ABB RAPID module: 000EB206

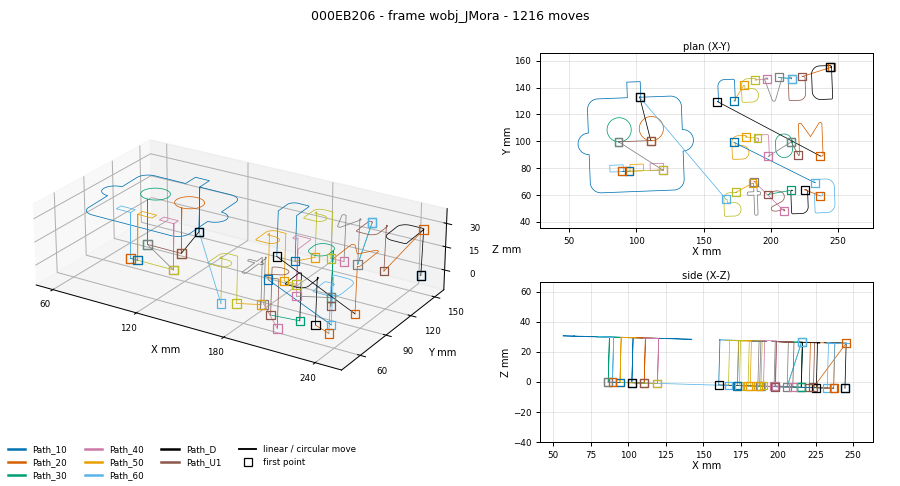
[picture p0: tool path of 000EB206 in frame wobj_JMora, 1216 of 1225 moves have a stored position in this frame; points joined in program order, loops and branches not executed]
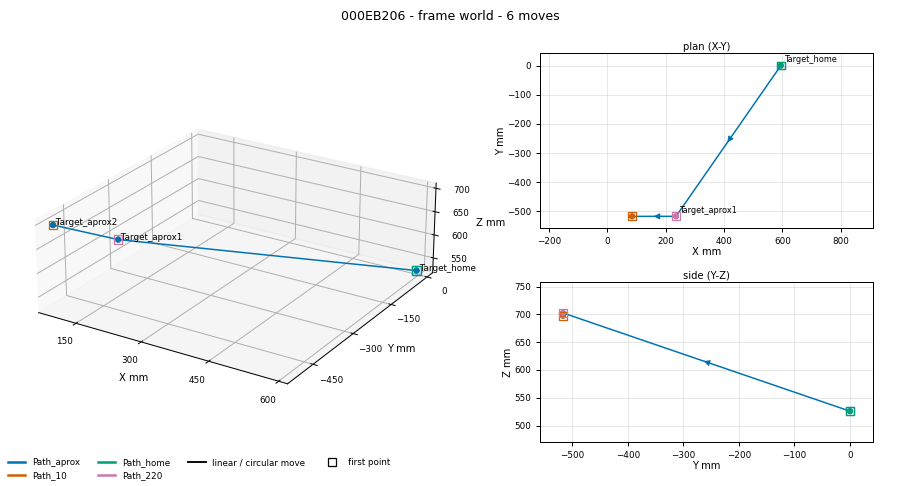
[picture p1: tool path of 000EB206 in frame world, 6 of 1225 moves have a stored position in this frame; points joined in program order, loops and branches not executed]
MODULE Module1
	PERS tooldata toolreal_fin:=[TRUE,[[75.2786,-1.94785,145.188],[1,0,0,0]],[1,[0,0,0],[1,0,0,0],0,0,0]];
    TASK PERS tooldata toolreal:=[TRUE,[[0,0,0],[1,0,0,0]],[-1,[0,0,0],[1,0,0,0],0,0,0]];

    CONST robtarget Target_home:=[[594.991189092,-0.007598177,525.862524879],[0.258822484,0.000002114,0.965924905,-0.000003007],[0,0,0,0],[9E+09,9E+09,9E+09,9E+09,9E+09,9E+09]];
    CONST robtarget Target_aprox1:=[[235.86399401,-516.605376424,702.653598227],[0,0.707106781,0.707106781,0],[0,0,0,0],[9E+09,9E+09,9E+09,9E+09,9E+09,9E+09]];
    CONST robtarget Target_aprox2:=[[85.598000009,-516.640000054,697.650000033],[0,0.707106781,0.707106781,0],[0,0,0,0],[9E+09,9E+09,9E+09,9E+09,9E+09,9E+09]];
    CONST robtarget Target_10:=[[244.458254265,155.289204222,-4.164726397],[0.692516726,0.060687774,-0.040025667,0.717729422],[-2,0,-1,0],[9E+09,9E+09,9E+09,9E+09,9E+09,9E+09]];
    CONST robtarget Target_20:=[[245.259577842,155.215414434,25.824478921],[0.692516726,0.060687774,-0.040025667,0.717729422],[-2,0,-1,0],[9E+09,9E+09,9E+09,9E+09,9E+09,9E+09]];
    CONST robtarget Target_30:=[[245.229089406,155.507196472,25.826011527],[0.692516726,0.060687774,-0.040025667,0.717729422],[-2,0,-1,0],[9E+09,9E+09,9E+09,9E+09,9E+09,9E+09]];
    CONST robtarget Target_40:=[[245.16107836,155.758507333,25.82844716],[0.692516726,0.060687774,-0.040025666,0.717729422],[-2,0,-1,0],[9E+09,9E+09,9E+09,9E+09,9E+09,9E+09]];
    CONST robtarget Target_50:=[[245.055544704,155.969347015,25.831785853],[0.692516726,0.060687774,-0.040025667,0.717729422],[-2,0,-1,0],[9E+09,9E+09,9E+09,9E+09,9E+09,9E+09]];
    CONST robtarget Target_60:=[[244.912488436,156.139715523,25.836027573],[0.692516726,0.060687774,-0.040025667,0.717729422],[-2,0,-1,0],[9E+09,9E+09,9E+09,9E+09,9E+09,9E+09]];
    CONST robtarget Target_70:=[[244.73190956,156.269612854,25.841172332],[0.692516726,0.060687774,-0.040025667,0.717729422],[-2,0,-1,0],[9E+09,9E+09,9E+09,9E+09,9E+09,9E+09]];
    CONST robtarget Target_80:=[[244.513808072,156.359039007,25.847220128],[0.692516726,0.060687774,-0.040025667,0.717729422],[-2,0,-1,0],[9E+09,9E+09,9E+09,9E+09,9E+09,9E+09]];
    CONST robtarget Target_90:=[[244.258183973,156.407993984,25.854170962],[0.692516726,0.060687774,-0.040025667,0.717729422],[-2,0,-1,0],[9E+09,9E+09,9E+09,9E+09,9E+09,9E+09]];
    CONST robtarget Target_100:=[[243.965037266,156.416477784,25.862024834],[0.692516726,0.060687774,-0.040025667,0.717729422],[-2,0,-1,0],[9E+09,9E+09,9E+09,9E+09,9E+09,9E+09]];
    CONST robtarget Target_110:=[[236.458451079,156.133651424,26.061907917],[0.692516726,0.060687774,-0.040025667,0.717729422],[-1,-1,0,0],[9E+09,9E+09,9E+09,9E+09,9E+09,9E+09]];
    CONST robtarget Target_120:=[[235.817178284,156.081173489,26.078913847],[0.692516726,0.060687774,-0.040025666,0.717729422],[-1,-1,0,0],[9E+09,9E+09,9E+09,9E+09,9E+09,9E+09]];
    CONST robtarget Target_130:=[[235.20337356,155.973097192,26.09504904],[0.692516726,0.060687774,-0.040025667,0.717729422],[-1,-1,0,0],[9E+09,9E+09,9E+09,9E+09,9E+09,9E+09]];
    CONST robtarget Target_140:=[[234.617036903,155.809422533,26.11031345],[0.692516726,0.060687774,-0.040025666,0.717729422],[-1,-1,0,0],[9E+09,9E+09,9E+09,9E+09,9E+09,9E+09]];
    CONST robtarget Target_150:=[[234.058168316,155.590149513,26.124707111],[0.692516726,0.060687774,-0.040025666,0.717729422],[-1,-1,0,0],[9E+09,9E+09,9E+09,9E+09,9E+09,9E+09]];
    CONST robtarget Target_160:=[[233.526767795,155.315278129,26.138230024],[0.692516726,0.060687774,-0.040025667,0.717729422],[-1,-1,0,0],[9E+09,9E+09,9E+09,9E+09,9E+09,9E+09]];
    CONST robtarget Target_170:=[[233.022835345,154.984808384,26.150882165],[0.692516726,0.060687774,-0.040025667,0.717729422],[-1,-1,0,0],[9E+09,9E+09,9E+09,9E+09,9E+09,9E+09]];
    CONST robtarget Target_180:=[[232.546370963,154.598740279,26.162663546],[0.692516726,0.060687774,-0.040025667,0.717729422],[-1,-1,0,0],[9E+09,9E+09,9E+09,9E+09,9E+09,9E+09]];
    CONST robtarget Target_190:=[[232.097374649,154.157073811,26.173574156],[0.692516726,0.060687774,-0.040025666,0.717729422],[-1,-1,0,0],[9E+09,9E+09,9E+09,9E+09,9E+09,9E+09]];
    CONST robtarget Target_200:=[[231.690855447,153.675997451,26.183252813],[0.692516726,0.060687774,-0.040025667,0.717729422],[-1,-1,0,0],[9E+09,9E+09,9E+09,9E+09,9E+09,9E+09]];
    CONST robtarget Target_210:=[[231.341822403,153.171699671,26.191338269],[0.692516726,0.060687774,-0.040025667,0.717729422],[-1,-1,0,0],[9E+09,9E+09,9E+09,9E+09,9E+09,9E+09]];
    CONST robtarget Target_220:=[[231.050275515,152.644180472,26.197830522],[0.692516726,0.060687774,-0.040025666,0.717729422],[-1,-1,0,0],[9E+09,9E+09,9E+09,9E+09,9E+09,9E+09]];
    CONST robtarget Target_230:=[[230.816214785,152.093439851,26.202729597],[0.692516726,0.060687774,-0.040025666,0.717729422],[-1,-1,0,0],[9E+09,9E+09,9E+09,9E+09,9E+09,9E+09]];
    CONST robtarget Target_240:=[[230.639640211,151.519477809,26.206035481],[0.692516726,0.060687774,-0.040025666,0.717729422],[-1,-1,0,0],[9E+09,9E+09,9E+09,9E+09,9E+09,9E+09]];
    CONST robtarget Target_250:=[[230.520551793,150.922294347,26.207748185],[0.692516726,0.060687774,-0.040025667,0.717729422],[-1,-1,0,0],[9E+09,9E+09,9E+09,9E+09,9E+09,9E+09]];
    CONST robtarget Target_260:=[[230.458949533,150.301889466,26.207867677],[0.692516726,0.060687774,-0.040025666,0.717729422],[-1,-1,0,0],[9E+09,9E+09,9E+09,9E+09,9E+09,9E+09]];
    CONST robtarget Target_270:=[[230.45483343,149.658263163,26.206394001],[0.692516726,0.060687774,-0.040025667,0.717729422],[-1,-1,0,0],[9E+09,9E+09,9E+09,9E+09,9E+09,9E+09]];
    CONST robtarget Target_280:=[[230.924700472,137.156756977,26.163078447],[0.692516726,0.060687774,-0.040025667,0.717729422],[-1,-1,0,0],[9E+09,9E+09,9E+09,9E+09,9E+09,9E+09]];
    CONST robtarget Target_290:=[[230.977088342,136.52469846,26.160123414],[0.692516726,0.060687774,-0.040025667,0.717729422],[-1,-1,0,0],[9E+09,9E+09,9E+09,9E+09,9E+09,9E+09]];
    CONST robtarget Target_300:=[[231.085779815,135.918195759,26.155726818],[0.692516726,0.060687774,-0.040025666,0.717729422],[-1,-1,0,0],[9E+09,9E+09,9E+09,9E+09,9E+09,9E+09]];
    CONST robtarget Target_310:=[[231.250774887,135.337248876,26.149888616],[0.692516726,0.060687774,-0.040025666,0.717729422],[-1,-1,0,0],[9E+09,9E+09,9E+09,9E+09,9E+09,9E+09]];
    CONST robtarget Target_320:=[[231.472073561,134.781857808,26.142608862],[0.692516726,0.060687774,-0.040025666,0.717729422],[-1,-1,0,0],[9E+09,9E+09,9E+09,9E+09,9E+09,9E+09]];
    CONST robtarget Target_330:=[[231.749675836,134.252022554,26.133887545],[0.692516726,0.060687774,-0.040025667,0.717729422],[-1,-1,0,0],[9E+09,9E+09,9E+09,9E+09,9E+09,9E+09]];
    CONST robtarget Target_340:=[[232.083581711,133.747743119,26.123724645],[0.692516726,0.060687774,-0.040025667,0.717729422],[-1,-1,0,0],[9E+09,9E+09,9E+09,9E+09,9E+09,9E+09]];
    CONST robtarget Target_350:=[[232.473791188,133.2690195,26.112120159],[0.692516726,0.060687774,-0.040025666,0.717729422],[-1,-1,0,0],[9E+09,9E+09,9E+09,9E+09,9E+09,9E+09]];
    CONST robtarget Target_360:=[[232.920304265,132.815851696,26.099074122],[0.692516726,0.060687774,-0.040025667,0.717729422],[-1,-1,0,0],[9E+09,9E+09,9E+09,9E+09,9E+09,9E+09]];
    CONST robtarget Target_370:=[[233.405590707,132.40450411,26.085094935],[0.692516726,0.060687774,-0.040025667,0.717729422],[-1,-1,0,0],[9E+09,9E+09,9E+09,9E+09,9E+09,9E+09]];
    CONST robtarget Target_380:=[[233.912120276,132.051241138,26.070691042],[0.692516726,0.060687774,-0.040025667,0.717729422],[-1,-1,0,0],[9E+09,9E+09,9E+09,9E+09,9E+09,9E+09]];
    CONST robtarget Target_390:=[[234.439892972,131.756062782,26.055862424],[0.692516726,0.060687774,-0.040025667,0.717729422],[-1,-1,0,0],[9E+09,9E+09,9E+09,9E+09,9E+09,9E+09]];
    CONST robtarget Target_400:=[[234.988908794,131.518969041,26.040609121],[0.692516726,0.060687774,-0.040025667,0.717729422],[-1,-1,0,0],[9E+09,9E+09,9E+09,9E+09,9E+09,9E+09]];
    CONST robtarget Target_410:=[[235.559167743,131.339959914,26.024931135],[0.692516726,0.060687774,-0.040025667,0.717729422],[-1,-1,0,0],[9E+09,9E+09,9E+09,9E+09,9E+09,9E+09]];
    CONST robtarget Target_420:=[[236.15066982,131.219035404,26.008828422],[0.692516726,0.060687774,-0.040025667,0.717729422],[-1,-1,0,0],[9E+09,9E+09,9E+09,9E+09,9E+09,9E+09]];
    CONST robtarget Target_430:=[[236.763415023,131.156195509,25.992301005],[0.692516726,0.060687774,-0.040025667,0.717729422],[-1,-1,0,0],[9E+09,9E+09,9E+09,9E+09,9E+09,9E+09]];
    CONST robtarget Target_440:=[[237.397403355,131.151440229,25.975348882],[0.692516726,0.060687774,-0.040025667,0.717729422],[-1,-1,0,0],[9E+09,9E+09,9E+09,9E+09,9E+09,9E+09]];
    CONST robtarget Target_530:=[[246.104713071,132.729344243,25.746568583],[0.692516726,0.060687774,-0.040025667,0.717729422],[-2,0,-1,0],[9E+09,9E+09,9E+09,9E+09,9E+09,9E+09]];
    CONST robtarget Target_510:=[[246.047258547,132.180375453,25.746753017],[0.692516726,0.060687774,-0.040025666,0.717729422],[-2,0,-1,0],[9E+09,9E+09,9E+09,9E+09,9E+09,9E+09]];
    CONST robtarget Target_520:=[[246.096213006,132.436093232,25.746074151],[0.692516726,0.060687774,-0.040025667,0.717729422],[-2,0,-1,0],[9E+09,9E+09,9E+09,9E+09,9E+09,9E+09]];
    CONST robtarget Target_540:=[[245.259577842,155.215414434,25.824478921],[0.692516726,0.060687774,-0.040025667,0.717729422],[-2,0,-1,0],[9E+09,9E+09,9E+09,9E+09,9E+09,9E+09]];
    CONST robtarget Target_500:=[[245.957849696,131.9621909,25.748605216],[0.692516726,0.060687774,-0.040025667,0.717729422],[-2,0,-1,0],[9E+09,9E+09,9E+09,9E+09,9E+09,9E+09]];
    CONST robtarget Target_450:=[[244.903989542,131.43426659,25.7754658],[0.692516726,0.060687774,-0.040025667,0.717729422],[-2,0,-1,0],[9E+09,9E+09,9E+09,9E+09,9E+09,9E+09]];
    CONST robtarget Target_460:=[[245.195670358,131.464784994,25.767747052],[0.692516726,0.060687774,-0.040025666,0.717729422],[-2,0,-1,0],[9E+09,9E+09,9E+09,9E+09,9E+09,9E+09]];
    CONST robtarget Target_480:=[[245.657668813,131.638421488,25.75582952],[0.692516726,0.060687774,-0.040025667,0.717729422],[-2,0,-1,0],[9E+09,9E+09,9E+09,9E+09,9E+09,9E+09]];
    CONST robtarget Target_490:=[[245.827986451,131.78153958,25.751630702],[0.692516726,0.060687774,-0.040025666,0.717729422],[-2,0,-1,0],[9E+09,9E+09,9E+09,9E+09,9E+09,9E+09]];
    CONST robtarget Target_470:=[[245.446896782,131.532836625,25.761201637],[0.692516726,0.060687774,-0.040025667,0.717729422],[-2,0,-1,0],[9E+09,9E+09,9E+09,9E+09,9E+09,9E+09]];
    CONST robtarget Target_550:=[[223.462258109,148.248946692,-3.621027841],[0.692516726,0.060687774,-0.040025667,0.717729422],[0,0,0,0],[9E+09,9E+09,9E+09,9E+09,9E+09,9E+09]];
    CONST robtarget Target_560:=[[224.263581686,148.175156905,26.368177477],[0.692516726,0.060687774,-0.040025667,0.717729422],[0,0,0,0],[9E+09,9E+09,9E+09,9E+09,9E+09,9E+09]];
    CONST robtarget Target_570:=[[224.556728395,148.166673106,26.360323594],[0.692516726,0.060687774,-0.040025666,0.717729422],[0,0,0,0],[9E+09,9E+09,9E+09,9E+09,9E+09,9E+09]];
    CONST robtarget Target_580:=[[224.812352494,148.117718127,26.353372782],[0.692516726,0.060687774,-0.040025666,0.717729422],[0,0,0,0],[9E+09,9E+09,9E+09,9E+09,9E+09,9E+09]];
    CONST robtarget Target_590:=[[225.03045398,148.028291975,26.347324964],[0.692516726,0.060687774,-0.040025666,0.717729422],[0,0,0,0],[9E+09,9E+09,9E+09,9E+09,9E+09,9E+09]];
    CONST robtarget Target_600:=[[225.211032857,147.898394643,26.342180217],[0.692516726,0.060687774,-0.040025667,0.717729422],[0,0,0,0],[9E+09,9E+09,9E+09,9E+09,9E+09,9E+09]];
    CONST robtarget Target_610:=[[225.354089124,147.728026137,26.337938485],[0.692516726,0.060687774,-0.040025666,0.717729422],[0,0,0,0],[9E+09,9E+09,9E+09,9E+09,9E+09,9E+09]];
    CONST robtarget Target_620:=[[225.459622781,147.517186454,26.334599803],[0.692516726,0.060687774,-0.040025666,0.717729422],[0,0,0,0],[9E+09,9E+09,9E+09,9E+09,9E+09,9E+09]];
    CONST robtarget Target_630:=[[225.527633827,147.265875592,26.33216417],[0.692516726,0.060687774,-0.040025667,0.717729422],[0,0,0,0],[9E+09,9E+09,9E+09,9E+09,9E+09,9E+09]];
    CONST robtarget Target_640:=[[225.558122263,146.974093555,26.330631564],[0.692516726,0.060687774,-0.040025667,0.717729422],[0,0,0,0],[9E+09,9E+09,9E+09,9E+09,9E+09,9E+09]];
    CONST robtarget Target_650:=[[225.981080782,135.720657872,26.291640359],[0.692516726,0.060687774,-0.040025667,0.717729422],[0,0,0,0],[9E+09,9E+09,9E+09,9E+09,9E+09,9E+09]];
    CONST robtarget Target_660:=[[225.977855815,135.204815501,26.290457267],[0.692516726,0.060687774,-0.040025666,0.717729422],[0,0,0,0],[9E+09,9E+09,9E+09,9E+09,9E+09,9E+09]];
    CONST robtarget Target_670:=[[225.928699575,134.707747724,26.290547695],[0.692516726,0.060687774,-0.040025667,0.717729422],[0,0,0,0],[9E+09,9E+09,9E+09,9E+09,9E+09,9E+09]];
    CONST robtarget Target_680:=[[225.833612059,134.229454546,26.291911598],[0.692516726,0.060687774,-0.040025666,0.717729422],[0,0,0,0],[9E+09,9E+09,9E+09,9E+09,9E+09,9E+09]];
    CONST robtarget Target_690:=[[225.69259327,133.769935961,26.294549011],[0.692516726,0.060687774,-0.040025666,0.717729422],[0,0,0,0],[9E+09,9E+09,9E+09,9E+09,9E+09,9E+09]];
    CONST robtarget Target_700:=[[225.505643208,133.329191973,26.298459921],[0.692516726,0.060687774,-0.040025666,0.717729422],[0,0,0,0],[9E+09,9E+09,9E+09,9E+09,9E+09,9E+09]];
    CONST robtarget Target_710:=[[225.272761871,132.907222579,26.30364434],[0.692516726,0.060687774,-0.040025667,0.717729422],[0,0,0,0],[9E+09,9E+09,9E+09,9E+09,9E+09,9E+09]];
    CONST robtarget Target_720:=[[224.99394926,132.504027783,26.310102235],[0.692516726,0.060687774,-0.040025666,0.717729422],[0,0,0,0],[9E+09,9E+09,9E+09,9E+09,9E+09,9E+09]];
    CONST robtarget Target_730:=[[224.669205374,132.119607582,26.317833638],[0.692516726,0.060687774,-0.040025666,0.717729422],[0,0,0,0],[9E+09,9E+09,9E+09,9E+09,9E+09,9E+09]];
    CONST robtarget Target_740:=[[224.310412375,131.766777849,26.326552577],[0.692516726,0.060687774,-0.040025666,0.717729422],[0,0,0,0],[9E+09,9E+09,9E+09,9E+09,9E+09,9E+09]];
    CONST robtarget Target_750:=[[223.929452421,131.458354456,26.33597309],[0.692516726,0.060687774,-0.040025666,0.717729422],[0,0,0,0],[9E+09,9E+09,9E+09,9E+09,9E+09,9E+09]];
    CONST robtarget Target_760:=[[223.526325513,131.194337404,26.346095188],[0.692516726,0.060687774,-0.040025667,0.717729422],[0,0,0,0],[9E+09,9E+09,9E+09,9E+09,9E+09,9E+09]];
    CONST robtarget Target_770:=[[223.101031652,130.974726695,26.356918848],[0.692516726,0.060687774,-0.040025667,0.717729422],[0,0,0,0],[9E+09,9E+09,9E+09,9E+09,9E+09,9E+09]];
    CONST robtarget Target_780:=[[222.653570836,130.799522325,26.368444082],[0.692516726,0.060687774,-0.040025667,0.717729422],[0,0,0,0],[9E+09,9E+09,9E+09,9E+09,9E+09,9E+09]];
    CONST robtarget Target_790:=[[222.183943066,130.668724296,26.38067089],[0.692516726,0.060687774,-0.040025667,0.717729422],[0,0,0,0],[9E+09,9E+09,9E+09,9E+09,9E+09,9E+09]];
    CONST robtarget Target_800:=[[221.692148341,130.582332609,26.393599271],[0.692516726,0.060687774,-0.040025667,0.717729422],[0,0,0,0],[9E+09,9E+09,9E+09,9E+09,9E+09,9E+09]];
    CONST robtarget Target_810:=[[221.178186662,130.540347262,26.407229226],[0.692516726,0.060687774,-0.040025667,0.717729422],[0,0,0,0],[9E+09,9E+09,9E+09,9E+09,9E+09,9E+09]];
    CONST robtarget Target_820:=[[214.919232528,130.304528053,26.573890744],[0.692516726,0.060687774,-0.040025667,0.717729422],[0,0,0,0],[9E+09,9E+09,9E+09,9E+09,9E+09,9E+09]];
    CONST robtarget Target_830:=[[214.626085821,130.313011855,26.581744605],[0.692516726,0.060687774,-0.040025666,0.717729422],[0,0,0,0],[9E+09,9E+09,9E+09,9E+09,9E+09,9E+09]];
    CONST robtarget Target_840:=[[214.370461724,130.36196683,26.588695461],[0.692516726,0.060687774,-0.040025666,0.717729422],[0,0,0,0],[9E+09,9E+09,9E+09,9E+09,9E+09,9E+09]];
    CONST robtarget Target_850:=[[214.152360235,130.451392985,26.594743235],[0.692516726,0.060687774,-0.040025666,0.717729422],[0,0,0,0],[9E+09,9E+09,9E+09,9E+09,9E+09,9E+09]];
    CONST robtarget Target_860:=[[213.971781358,130.581290314,26.599888004],[0.692516726,0.060687774,-0.040025667,0.717729422],[0,0,0,0],[9E+09,9E+09,9E+09,9E+09,9E+09,9E+09]];
    CONST robtarget Target_870:=[[213.828725091,130.751658823,26.604129713],[0.692516726,0.060687774,-0.040025666,0.717729422],[0,0,0,0],[9E+09,9E+09,9E+09,9E+09,9E+09,9E+09]];
    CONST robtarget Target_880:=[[213.723191435,130.962498507,26.607468396],[0.692516726,0.060687774,-0.040025666,0.717729422],[0,0,0,0],[9E+09,9E+09,9E+09,9E+09,9E+09,9E+09]];
    CONST robtarget Target_890:=[[213.655180388,131.213809365,26.609904051],[0.692516726,0.060687774,-0.040025667,0.717729422],[0,0,0,0],[9E+09,9E+09,9E+09,9E+09,9E+09,9E+09]];
    CONST robtarget Target_900:=[[213.624691952,131.505591403,26.611436657],[0.692516726,0.060687774,-0.040025667,0.717729422],[0,0,0,0],[9E+09,9E+09,9E+09,9E+09,9E+09,9E+09]];
    CONST robtarget Target_910:=[[213.061007863,146.503238589,26.663400906],[0.692516726,0.060687774,-0.040025667,0.717729422],[0,0,0,0],[9E+09,9E+09,9E+09,9E+09,9E+09,9E+09]];
    CONST robtarget Target_920:=[[213.069507929,146.796489599,26.663895338],[0.692516726,0.060687774,-0.040025667,0.717729422],[0,0,0,0],[9E+09,9E+09,9E+09,9E+09,9E+09,9E+09]];
    CONST robtarget Target_930:=[[213.118462388,147.052207381,26.66321645],[0.692516726,0.060687774,-0.040025666,0.717729422],[0,0,0,0],[9E+09,9E+09,9E+09,9E+09,9E+09,9E+09]];
    CONST robtarget Target_940:=[[213.207871239,147.270391931,26.661364273],[0.692516726,0.060687774,-0.040025667,0.717729422],[0,0,0,0],[9E+09,9E+09,9E+09,9E+09,9E+09,9E+09]];
    CONST robtarget Target_950:=[[213.337734484,147.451043254,26.658338765],[0.692516726,0.060687774,-0.040025666,0.717729422],[0,0,0,0],[9E+09,9E+09,9E+09,9E+09,9E+09,9E+09]];
    CONST robtarget Target_960:=[[213.508052121,147.594161345,26.654139969],[0.692516726,0.060687774,-0.040025667,0.717729422],[0,0,0,0],[9E+09,9E+09,9E+09,9E+09,9E+09,9E+09]];
    CONST robtarget Target_970:=[[213.718824152,147.699746206,26.648767852],[0.692516726,0.060687774,-0.040025667,0.717729422],[0,0,0,0],[9E+09,9E+09,9E+09,9E+09,9E+09,9E+09]];
    CONST robtarget Target_980:=[[213.970050576,147.76779784,26.642222415],[0.692516726,0.060687774,-0.040025666,0.717729422],[0,0,0,0],[9E+09,9E+09,9E+09,9E+09,9E+09,9E+09]];
    CONST robtarget Target_990:=[[214.261731393,147.798316241,26.634503689],[0.692516726,0.060687774,-0.040025667,0.717729422],[0,0,0,0],[9E+09,9E+09,9E+09,9E+09,9E+09,9E+09]];
    CONST robtarget Target_1000:=[[214.554878101,147.789832442,26.626649806],[0.692516726,0.060687774,-0.040025666,0.717729422],[0,0,0,0],[9E+09,9E+09,9E+09,9E+09,9E+09,9E+09]];
    CONST robtarget Target_1010:=[[214.8105022,147.740877464,26.619698994],[0.692516726,0.060687774,-0.040025666,0.717729422],[0,0,0,0],[9E+09,9E+09,9E+09,9E+09,9E+09,9E+09]];
    CONST robtarget Target_1020:=[[215.028603686,147.651451311,26.613651176],[0.692516726,0.060687774,-0.040025666,0.717729422],[0,0,0,0],[9E+09,9E+09,9E+09,9E+09,9E+09,9E+09]];
    CONST robtarget Target_1030:=[[215.209182564,147.52155398,26.608506429],[0.692516726,0.060687774,-0.040025667,0.717729422],[0,0,0,0],[9E+09,9E+09,9E+09,9E+09,9E+09,9E+09]];
    CONST robtarget Target_1040:=[[215.35223883,147.351185473,26.604264698],[0.692516726,0.060687774,-0.040025666,0.717729422],[0,0,0,0],[9E+09,9E+09,9E+09,9E+09,9E+09,9E+09]];
    CONST robtarget Target_1050:=[[215.457772487,147.14034579,26.600926016],[0.692516726,0.060687774,-0.040025666,0.717729422],[0,0,0,0],[9E+09,9E+09,9E+09,9E+09,9E+09,9E+09]];
    CONST robtarget Target_1060:=[[215.525783533,146.889034929,26.598490382],[0.692516726,0.060687774,-0.040025667,0.717729422],[0,0,0,0],[9E+09,9E+09,9E+09,9E+09,9E+09,9E+09]];
    CONST robtarget Target_1070:=[[215.55627197,146.597252891,26.596957776],[0.692516726,0.060687774,-0.040025667,0.717729422],[0,0,0,0],[9E+09,9E+09,9E+09,9E+09,9E+09,9E+09]];
    CONST robtarget Target_1080:=[[205.974615496,147.590063121,-3.155372239],[0.692516726,0.060687774,-0.040025667,0.717729422],[0,0,0,0],[9E+09,9E+09,9E+09,9E+09,9E+09,9E+09]];
    CONST robtarget Target_1090:=[[206.775939073,147.516273333,26.833833079],[0.692516726,0.060687774,-0.040025667,0.717729422],[0,0,0,0],[9E+09,9E+09,9E+09,9E+09,9E+09,9E+09]];
    CONST robtarget Target_1100:=[[207.018522887,147.502629685,26.827317561],[0.692516726,0.060687774,-0.040025666,0.717729422],[0,0,0,0],[9E+09,9E+09,9E+09,9E+09,9E+09,9E+09]];
    CONST robtarget Target_1110:=[[207.247221507,147.442895875,26.821059664],[0.692516726,0.060687774,-0.040025666,0.717729422],[0,0,0,0],[9E+09,9E+09,9E+09,9E+09,9E+09,9E+09]];
    CONST robtarget Target_1120:=[[207.462034933,147.337071905,26.815059401],[0.692516726,0.060687774,-0.040025666,0.717729422],[0,0,0,0],[9E+09,9E+09,9E+09,9E+09,9E+09,9E+09]];
    CONST robtarget Target_1130:=[[207.662963164,147.185157777,26.809316704],[0.692516726,0.060687774,-0.040025666,0.717729422],[0,0,0,0],[9E+09,9E+09,9E+09,9E+09,9E+09,9E+09]];
    CONST robtarget Target_1140:=[[207.833873307,147.000866706,26.804296471],[0.692516726,0.060687774,-0.040025667,0.717729422],[0,0,0,0],[9E+09,9E+09,9E+09,9E+09,9E+09,9E+09]];
    CONST robtarget Target_1150:=[[207.958632467,146.797911914,26.800463466],[0.692516726,0.060687774,-0.040025666,0.717729422],[0,0,0,0],[9E+09,9E+09,9E+09,9E+09,9E+09,9E+09]];
    CONST robtarget Target_1160:=[[208.037240646,146.576293398,26.797817744],[0.692516726,0.060687774,-0.040025666,0.717729422],[0,0,0,0],[9E+09,9E+09,9E+09,9E+09,9E+09,9E+09]];
    CONST robtarget Target_1170:=[[208.069697841,146.336011159,26.796359239],[0.692516726,0.060687774,-0.040025667,0.717729422],[0,0,0,0],[9E+09,9E+09,9E+09,9E+09,9E+09,9E+09]];
    CONST robtarget Target_1180:=[[208.056331156,146.137616545,26.796228232],[0.692516726,0.060687774,-0.040025666,0.717729422],[0,0,0,0],[9E+09,9E+09,9E+09,9E+09,9E+09,9E+09]];
    CONST robtarget Target_1190:=[[208.002158545,145.91685385,26.797132549],[0.692516726,0.060687774,-0.040025666,0.717729422],[0,0,0,0],[9E+09,9E+09,9E+09,9E+09,9E+09,9E+09]];
    CONST robtarget Target_1200:=[[203.652235422,130.900721267,26.876416368],[0.692516726,0.060687774,-0.040025666,0.717729422],[0,0,0,0],[9E+09,9E+09,9E+09,9E+09,9E+09,9E+09]];
    CONST robtarget Target_1210:=[[203.564392561,130.658184821,26.878166804],[0.692516726,0.060687774,-0.040025667,0.717729422],[0,0,0,0],[9E+09,9E+09,9E+09,9E+09,9E+09,9E+09]];
    CONST robtarget Target_1220:=[[203.458457537,130.44686362,26.880477464],[0.692516726,0.060687774,-0.040025667,0.717729422],[0,0,0,0],[9E+09,9E+09,9E+09,9E+09,9E+09,9E+09]];
    CONST robtarget Target_1230:=[[203.334430353,130.266757664,26.883348351],[0.692516726,0.060687774,-0.040025666,0.717729422],[0,0,0,0],[9E+09,9E+09,9E+09,9E+09,9E+09,9E+09]];
    CONST robtarget Target_1240:=[[203.192311005,130.11786695,26.886779495],[0.692516726,0.060687774,-0.040025667,0.717729422],[0,0,0,0],[9E+09,9E+09,9E+09,9E+09,9E+09,9E+09]];
    CONST robtarget Target_1250:=[[203.032099496,130.000191481,26.890770865],[0.692516726,0.060687774,-0.040025667,0.717729422],[0,0,0,0],[9E+09,9E+09,9E+09,9E+09,9E+09,9E+09]];
    CONST robtarget Target_1260:=[[202.853795825,129.913731256,26.895322471],[0.692516726,0.060687774,-0.040025667,0.717729422],[0,0,0,0],[9E+09,9E+09,9E+09,9E+09,9E+09,9E+09]];
    CONST robtarget Target_1270:=[[202.657399992,129.858486276,26.900434314],[0.692516726,0.060687774,-0.040025667,0.717729422],[0,0,0,0],[9E+09,9E+09,9E+09,9E+09,9E+09,9E+09]];
    CONST robtarget Target_1280:=[[202.442911997,129.834456539,26.906106393],[0.692516726,0.060687774,-0.040025667,0.717729422],[0,0,0,0],[9E+09,9E+09,9E+09,9E+09,9E+09,9E+09]];
    CONST robtarget Target_1290:=[[202.222341078,129.84242,26.91201972],[0.692516726,0.060687774,-0.040025666,0.717729422],[0,0,0,0],[9E+09,9E+09,9E+09,9E+09,9E+09,9E+09]];
    CONST robtarget Target_1300:=[[202.018093409,129.883546331,26.917578503],[0.692516726,0.060687774,-0.040025667,0.717729422],[0,0,0,0],[9E+09,9E+09,9E+09,9E+09,9E+09,9E+09]];
    CONST robtarget Target_1310:=[[201.830168991,129.95783554,26.9227827],[0.692516726,0.060687774,-0.040025666,0.717729422],[0,0,0,0],[9E+09,9E+09,9E+09,9E+09,9E+09,9E+09]];
    CONST robtarget Target_1320:=[[201.658567821,130.065287622,26.927632343],[0.692516726,0.060687774,-0.040025666,0.717729422],[0,0,0,0],[9E+09,9E+09,9E+09,9E+09,9E+09,9E+09]];
    CONST robtarget Target_1330:=[[201.503289901,130.205902577,26.93212742],[0.692516726,0.060687774,-0.040025666,0.717729422],[0,0,0,0],[9E+09,9E+09,9E+09,9E+09,9E+09,9E+09]];
    CONST robtarget Target_1340:=[[201.364335231,130.379680405,26.936267944],[0.692516726,0.060687774,-0.040025667,0.717729422],[0,0,0,0],[9E+09,9E+09,9E+09,9E+09,9E+09,9E+09]];
    CONST robtarget Target_1350:=[[201.24170381,130.586621109,26.940053891],[0.692516726,0.060687774,-0.040025667,0.717729422],[0,0,0,0],[9E+09,9E+09,9E+09,9E+09,9E+09,9E+09]];
    CONST robtarget Target_1360:=[[201.135395639,130.826724686,26.943485274],[0.692516726,0.060687774,-0.040025667,0.717729422],[0,0,0,0],[9E+09,9E+09,9E+09,9E+09,9E+09,9E+09]];
    CONST robtarget Target_1370:=[[195.671395086,145.452266503,27.12547236],[0.692516726,0.060687774,-0.040025667,0.717729422],[0,0,0,0],[9E+09,9E+09,9E+09,9E+09,9E+09,9E+09]];
    CONST robtarget Target_1380:=[[195.600804491,145.668328483,27.127890199],[0.692516726,0.060687774,-0.040025667,0.717729422],[0,0,0,0],[9E+09,9E+09,9E+09,9E+09,9E+09,9E+09]];
    CONST robtarget Target_1390:=[[195.572583442,145.865156193,27.129128581],[0.692516726,0.060687774,-0.040025667,0.717729422],[0,0,0,0],[9E+09,9E+09,9E+09,9E+09,9E+09,9E+09]];
    CONST robtarget Target_1400:=[[195.581591648,146.153544169,27.129597469],[0.692516726,0.060687774,-0.040025667,0.717729422],[0,0,0,0],[9E+09,9E+09,9E+09,9E+09,9E+09,9E+09]];
    CONST robtarget Target_1410:=[[195.631679624,146.405073435,27.128877998],[0.692516726,0.060687774,-0.040025667,0.717729422],[0,0,0,0],[9E+09,9E+09,9E+09,9E+09,9E+09,9E+09]];
    CONST robtarget Target_1420:=[[195.722847369,146.619743992,27.126970165],[0.692516726,0.060687774,-0.040025667,0.717729422],[0,0,0,0],[9E+09,9E+09,9E+09,9E+09,9E+09,9E+09]];
    CONST robtarget Target_1430:=[[195.855094885,146.79755584,27.123873962],[0.692516726,0.060687774,-0.040025666,0.717729422],[0,0,0,0],[9E+09,9E+09,9E+09,9E+09,9E+09,9E+09]];
    CONST robtarget Target_1440:=[[196.028422171,146.938508975,27.11958942],[0.692516726,0.060687774,-0.040025667,0.717729422],[0,0,0,0],[9E+09,9E+09,9E+09,9E+09,9E+09,9E+09]];
    CONST robtarget Target_1450:=[[196.242829227,147.0426034,27.114116507],[0.692516726,0.060687774,-0.040025667,0.717729422],[0,0,0,0],[9E+09,9E+09,9E+09,9E+09,9E+09,9E+09]];
    CONST robtarget Target_1460:=[[196.498316052,147.109839116,27.107455233],[0.692516726,0.060687774,-0.040025667,0.717729422],[0,0,0,0],[9E+09,9E+09,9E+09,9E+09,9E+09,9E+09]];
    CONST robtarget Target_1470:=[[196.794882648,147.140216122,27.099605599],[0.692516726,0.060687774,-0.040025667,0.717729422],[0,0,0,0],[9E+09,9E+09,9E+09,9E+09,9E+09,9E+09]];
    CONST robtarget Target_1480:=[[197.014368912,147.135141106,27.093728339],[0.692516726,0.060687774,-0.040025666,0.717729422],[0,0,0,0],[9E+09,9E+09,9E+09,9E+09,9E+09,9E+09]];
    CONST robtarget Target_1490:=[[197.215362618,147.102680093,27.088277857],[0.692516726,0.060687774,-0.040025666,0.717729422],[0,0,0,0],[9E+09,9E+09,9E+09,9E+09,9E+09,9E+09]];
    CONST robtarget Target_1500:=[[197.397863764,147.042833091,27.083254086],[0.692516726,0.060687774,-0.040025667,0.717729422],[0,0,0,0],[9E+09,9E+09,9E+09,9E+09,9E+09,9E+09]];
    CONST robtarget Target_1510:=[[197.561872353,146.955600097,27.078657059],[0.692516726,0.060687774,-0.040025666,0.717729422],[0,0,0,0],[9E+09,9E+09,9E+09,9E+09,9E+09,9E+09]];
    CONST robtarget Target_1520:=[[197.707388383,146.840981108,27.074486799],[0.692516726,0.060687774,-0.040025667,0.717729422],[0,0,0,0],[9E+09,9E+09,9E+09,9E+09,9E+09,9E+09]];
    CONST robtarget Target_1530:=[[197.834411855,146.69897613,27.07074326],[0.692516726,0.060687774,-0.040025666,0.717729422],[0,0,0,0],[9E+09,9E+09,9E+09,9E+09,9E+09,9E+09]];
    CONST robtarget Target_1540:=[[197.942942768,146.529585157,27.067426487],[0.692516726,0.060687774,-0.040025667,0.717729422],[0,0,0,0],[9E+09,9E+09,9E+09,9E+09,9E+09,9E+09]];
    CONST robtarget Target_1550:=[[198.032981123,146.332808193,27.064536448],[0.692516726,0.060687774,-0.040025667,0.717729422],[0,0,0,0],[9E+09,9E+09,9E+09,9E+09,9E+09,9E+09]];
    CONST robtarget Target_1560:=[[197.231657546,146.406597981,-2.92466887],[0.692516726,0.060687774,-0.040025667,0.717729422],[0,0,0,0],[9E+09,9E+09,9E+09,9E+09,9E+09,9E+09]];
    CONST robtarget Target_1570:=[[188.51308754,145.682325596,-2.693487292],[0.692516726,0.060687774,-0.040025667,0.717729422],[0,0,0,0],[9E+09,9E+09,9E+09,9E+09,9E+09,9E+09]];
    CONST robtarget Target_1580:=[[189.314411117,145.608535808,27.295718026],[0.692516726,0.060687774,-0.040025667,0.717729422],[0,0,0,0],[9E+09,9E+09,9E+09,9E+09,9E+09,9E+09]];
    CONST robtarget Target_1590:=[[189.28392268,145.900317845,27.297250632],[0.692516726,0.060687774,-0.040025667,0.717729422],[0,0,0,0],[9E+09,9E+09,9E+09,9E+09,9E+09,9E+09]];
    CONST robtarget Target_1600:=[[189.215911634,146.151628707,27.299686265],[0.692516726,0.060687774,-0.040025666,0.717729422],[0,0,0,0],[9E+09,9E+09,9E+09,9E+09,9E+09,9E+09]];
    CONST robtarget Target_1610:=[[189.110377977,146.36246839,27.303024947],[0.692516726,0.060687774,-0.040025666,0.717729422],[0,0,0,0],[9E+09,9E+09,9E+09,9E+09,9E+09,9E+09]];
    CONST robtarget Target_1620:=[[188.96732171,146.532836896,27.307266678],[0.692516726,0.060687774,-0.040025667,0.717729422],[0,0,0,0],[9E+09,9E+09,9E+09,9E+09,9E+09,9E+09]];
    CONST robtarget Target_1630:=[[188.786742833,146.662734228,27.312411425],[0.692516726,0.060687774,-0.040025666,0.717729422],[0,0,0,0],[9E+09,9E+09,9E+09,9E+09,9E+09,9E+09]];
    CONST robtarget Target_1640:=[[188.568641346,146.75216038,27.318459243],[0.692516726,0.060687774,-0.040025666,0.717729422],[0,0,0,0],[9E+09,9E+09,9E+09,9E+09,9E+09,9E+09]];
    CONST robtarget Target_1650:=[[188.313017248,146.801115359,27.325410055],[0.692516726,0.060687774,-0.040025666,0.717729422],[0,0,0,0],[9E+09,9E+09,9E+09,9E+09,9E+09,9E+09]];
    CONST robtarget Target_1660:=[[188.01987054,146.809599158,27.333263939],[0.692516726,0.060687774,-0.040025667,0.717729422],[0,0,0,0],[9E+09,9E+09,9E+09,9E+09,9E+09,9E+09]];
    CONST robtarget Target_1670:=[[183.029342326,146.621570553,27.466150198],[0.692516726,0.060687774,-0.040025667,0.717729422],[0,0,0,0],[9E+09,9E+09,9E+09,9E+09,9E+09,9E+09]];
    CONST robtarget Target_1680:=[[182.515380648,146.579585206,27.479780153],[0.692516726,0.060687774,-0.040025667,0.717729422],[0,0,0,0],[9E+09,9E+09,9E+09,9E+09,9E+09,9E+09]];
    CONST robtarget Target_1690:=[[182.023585924,146.493193519,27.492708535],[0.692516726,0.060687774,-0.040025667,0.717729422],[0,0,0,0],[9E+09,9E+09,9E+09,9E+09,9E+09,9E+09]];
    CONST robtarget Target_1700:=[[181.553958153,146.36239549,27.504935342],[0.692516726,0.060687774,-0.040025667,0.717729422],[0,0,0,0],[9E+09,9E+09,9E+09,9E+09,9E+09,9E+09]];
    CONST robtarget Target_1710:=[[181.106497337,146.187191121,27.516460576],[0.692516726,0.060687774,-0.040025667,0.717729422],[0,0,0,0],[9E+09,9E+09,9E+09,9E+09,9E+09,9E+09]];
    CONST robtarget Target_1720:=[[180.681203475,145.967580411,27.527284237],[0.692516726,0.060687774,-0.040025667,0.717729422],[0,0,0,0],[9E+09,9E+09,9E+09,9E+09,9E+09,9E+09]];
    CONST robtarget Target_1730:=[[180.278076568,145.70356336,27.537406312],[0.692516726,0.060687774,-0.040025666,0.717729422],[0,0,0,0],[9E+09,9E+09,9E+09,9E+09,9E+09,9E+09]];
    CONST robtarget Target_1740:=[[179.897116615,145.395139968,27.546826825],[0.692516726,0.060687774,-0.040025666,0.717729422],[0,0,0,0],[9E+09,9E+09,9E+09,9E+09,9E+09,9E+09]];
    CONST robtarget Target_1750:=[[179.538323615,145.042310235,27.555545764],[0.692516726,0.060687774,-0.040025666,0.717729422],[0,0,0,0],[9E+09,9E+09,9E+09,9E+09,9E+09,9E+09]];
    CONST robtarget Target_1760:=[[179.21357973,144.657890034,27.563277168],[0.692516726,0.060687774,-0.040025666,0.717729422],[0,0,0,0],[9E+09,9E+09,9E+09,9E+09,9E+09,9E+09]];
    CONST robtarget Target_1770:=[[178.934767119,144.254695235,27.569735085],[0.692516726,0.060687774,-0.040025667,0.717729422],[0,0,0,0],[9E+09,9E+09,9E+09,9E+09,9E+09,9E+09]];
    CONST robtarget Target_1780:=[[178.701885782,143.832725843,27.574919482],[0.692516726,0.060687774,-0.040025666,0.717729422],[0,0,0,0],[9E+09,9E+09,9E+09,9E+09,9E+09,9E+09]];
    CONST robtarget Target_1790:=[[178.514935719,143.391981856,27.578830392],[0.692516726,0.060687774,-0.040025666,0.717729422],[0,0,0,0],[9E+09,9E+09,9E+09,9E+09,9E+09,9E+09]];
    CONST robtarget Target_1800:=[[178.373916929,142.932463271,27.581467804],[0.692516726,0.060687774,-0.040025666,0.717729422],[0,0,0,0],[9E+09,9E+09,9E+09,9E+09,9E+09,9E+09]];
    CONST robtarget Target_1810:=[[178.278829415,142.45417009,27.58283173],[0.692516726,0.060687774,-0.040025667,0.717729422],[0,0,0,0],[9E+09,9E+09,9E+09,9E+09,9E+09,9E+09]];
    CONST robtarget Target_1820:=[[178.229673174,141.957102316,27.582922136],[0.692516726,0.060687774,-0.040025666,0.717729422],[0,0,0,0],[9E+09,9E+09,9E+09,9E+09,9E+09,9E+09]];
    CONST robtarget Target_1830:=[[178.226448208,141.441259943,27.581739066],[0.692516726,0.060687774,-0.040025667,0.717729422],[0,0,0,0],[9E+09,9E+09,9E+09,9E+09,9E+09,9E+09]];
    CONST robtarget Target_1840:=[[178.649406727,130.18782426,27.54274786],[0.692516726,0.060687774,-0.040025667,0.717729422],[0,0,0,0],[9E+09,9E+09,9E+09,9E+09,9E+09,9E+09]];
    CONST robtarget Target_1850:=[[178.679895162,129.896042223,27.541215254],[0.692516726,0.060687774,-0.040025667,0.717729422],[0,0,0,0],[9E+09,9E+09,9E+09,9E+09,9E+09,9E+09]];
    CONST robtarget Target_1860:=[[178.747906209,129.644731364,27.538779599],[0.692516726,0.060687774,-0.040025666,0.717729422],[0,0,0,0],[9E+09,9E+09,9E+09,9E+09,9E+09,9E+09]];
    CONST robtarget Target_1870:=[[178.853439865,129.43389168,27.535440917],[0.692516726,0.060687774,-0.040025666,0.717729422],[0,0,0,0],[9E+09,9E+09,9E+09,9E+09,9E+09,9E+09]];
    CONST robtarget Target_1880:=[[178.996496132,129.263523172,27.531199208],[0.692516726,0.060687774,-0.040025667,0.717729422],[0,0,0,0],[9E+09,9E+09,9E+09,9E+09,9E+09,9E+09]];
    CONST robtarget Target_1890:=[[179.177075009,129.133625843,27.526054439],[0.692516726,0.060687774,-0.040025666,0.717729422],[0,0,0,0],[9E+09,9E+09,9E+09,9E+09,9E+09,9E+09]];
    CONST robtarget Target_1900:=[[179.395176498,129.044199688,27.520006665],[0.692516726,0.060687774,-0.040025666,0.717729422],[0,0,0,0],[9E+09,9E+09,9E+09,9E+09,9E+09,9E+09]];
    CONST robtarget Target_1910:=[[179.650800595,128.995244712,27.513055808],[0.692516726,0.060687774,-0.040025666,0.717729422],[0,0,0,0],[9E+09,9E+09,9E+09,9E+09,9E+09,9E+09]];
    CONST robtarget Target_1920:=[[179.943947303,128.98676091,27.505201947],[0.692516726,0.060687774,-0.040025667,0.717729422],[0,0,0,0],[9E+09,9E+09,9E+09,9E+09,9E+09,9E+09]];
    CONST robtarget Target_1930:=[[186.182107569,129.221796667,27.339094123],[0.692516726,0.060687774,-0.040025667,0.717729422],[0,0,0,0],[9E+09,9E+09,9E+09,9E+09,9E+09,9E+09]];
    CONST robtarget Target_1940:=[[186.696069248,129.263782014,27.325464167],[0.692516726,0.060687774,-0.040025667,0.717729422],[0,0,0,0],[9E+09,9E+09,9E+09,9E+09,9E+09,9E+09]];
    CONST robtarget Target_1950:=[[187.187863972,129.350173701,27.312535786],[0.692516726,0.060687774,-0.040025667,0.717729422],[0,0,0,0],[9E+09,9E+09,9E+09,9E+09,9E+09,9E+09]];
    CONST robtarget Target_1960:=[[187.657491742,129.48097173,27.300308978],[0.692516726,0.060687774,-0.040025667,0.717729422],[0,0,0,0],[9E+09,9E+09,9E+09,9E+09,9E+09,9E+09]];
    CONST robtarget Target_1970:=[[188.104952558,129.656176099,27.288783744],[0.692516726,0.060687774,-0.040025667,0.717729422],[0,0,0,0],[9E+09,9E+09,9E+09,9E+09,9E+09,9E+09]];
    CONST robtarget Target_1980:=[[188.530246421,129.875786809,27.277960084],[0.692516726,0.060687774,-0.040025667,0.717729422],[0,0,0,0],[9E+09,9E+09,9E+09,9E+09,9E+09,9E+09]];
    CONST robtarget Target_1990:=[[188.933373328,130.139803861,27.267837987],[0.692516726,0.060687774,-0.040025666,0.717729422],[0,0,0,0],[9E+09,9E+09,9E+09,9E+09,9E+09,9E+09]];
    CONST robtarget Target_2000:=[[189.314333281,130.448227253,27.258417474],[0.692516726,0.060687774,-0.040025666,0.717729422],[0,0,0,0],[9E+09,9E+09,9E+09,9E+09,9E+09,9E+09]];
    CONST robtarget Target_2010:=[[189.673126281,130.801056986,27.249698534],[0.692516726,0.060687774,-0.040025666,0.717729422],[0,0,0,0],[9E+09,9E+09,9E+09,9E+09,9E+09,9E+09]];
    CONST robtarget Target_2020:=[[189.997870166,131.185477188,27.241967131],[0.692516726,0.060687774,-0.040025666,0.717729422],[0,0,0,0],[9E+09,9E+09,9E+09,9E+09,9E+09,9E+09]];
    CONST robtarget Target_2030:=[[190.276682777,131.588671984,27.235509236],[0.692516726,0.060687774,-0.040025667,0.717729422],[0,0,0,0],[9E+09,9E+09,9E+09,9E+09,9E+09,9E+09]];
    CONST robtarget Target_2040:=[[190.509564114,132.010641378,27.230324817],[0.692516726,0.060687774,-0.040025666,0.717729422],[0,0,0,0],[9E+09,9E+09,9E+09,9E+09,9E+09,9E+09]];
    CONST robtarget Target_2050:=[[190.696514177,132.451385366,27.226413907],[0.692516726,0.060687774,-0.040025666,0.717729422],[0,0,0,0],[9E+09,9E+09,9E+09,9E+09,9E+09,9E+09]];
    CONST robtarget Target_2060:=[[190.837532966,132.91090395,27.223776495],[0.692516726,0.060687774,-0.040025666,0.717729422],[0,0,0,0],[9E+09,9E+09,9E+09,9E+09,9E+09,9E+09]];
    CONST robtarget Target_2070:=[[190.932620481,133.389197129,27.222412591],[0.692516726,0.060687774,-0.040025667,0.717729422],[0,0,0,0],[9E+09,9E+09,9E+09,9E+09,9E+09,9E+09]];
    CONST robtarget Target_2080:=[[190.981776722,133.886264906,27.222322163],[0.692516726,0.060687774,-0.040025666,0.717729422],[0,0,0,0],[9E+09,9E+09,9E+09,9E+09,9E+09,9E+09]];
    CONST robtarget Target_2090:=[[190.985001688,134.402107276,27.223505255],[0.692516726,0.060687774,-0.040025667,0.717729422],[0,0,0,0],[9E+09,9E+09,9E+09,9E+09,9E+09,9E+09]];
    CONST robtarget Target_2100:=[[190.962335209,134.73682172,27.224934493],[0.692516726,0.060687774,-0.040025667,0.717729422],[0,0,0,0],[9E+09,9E+09,9E+09,9E+09,9E+09,9E+09]];
    CONST robtarget Target_2110:=[[190.919744554,135.064926865,27.226879838],[0.692516726,0.060687774,-0.040025666,0.717729422],[0,0,0,0],[9E+09,9E+09,9E+09,9E+09,9E+09,9E+09]];
    CONST robtarget Target_2120:=[[190.857229723,135.386422708,27.229341315],[0.692516726,0.060687774,-0.040025666,0.717729422],[0,0,0,0],[9E+09,9E+09,9E+09,9E+09,9E+09,9E+09]];
    CONST robtarget Target_2130:=[[190.774790718,135.701309253,27.23231891],[0.692516726,0.060687774,-0.040025666,0.717729422],[0,0,0,0],[9E+09,9E+09,9E+09,9E+09,9E+09,9E+09]];
    CONST robtarget Target_2140:=[[190.672427537,136.009586495,27.235812637],[0.692516726,0.060687774,-0.040025667,0.717729422],[0,0,0,0],[9E+09,9E+09,9E+09,9E+09,9E+09,9E+09]];
    CONST robtarget Target_2150:=[[190.55014018,136.311254438,27.239822471],[0.692516726,0.060687774,-0.040025667,0.717729422],[0,0,0,0],[9E+09,9E+09,9E+09,9E+09,9E+09,9E+09]];
    CONST robtarget Target_2160:=[[190.407928646,136.606313081,27.244348425],[0.692516726,0.060687774,-0.040025667,0.717729422],[0,0,0,0],[9E+09,9E+09,9E+09,9E+09,9E+09,9E+09]];
    CONST robtarget Target_2170:=[[190.245792939,136.894762425,27.249390499],[0.692516726,0.060687774,-0.040025667,0.717729422],[0,0,0,0],[9E+09,9E+09,9E+09,9E+09,9E+09,9E+09]];
    CONST robtarget Target_2180:=[[190.049412796,137.187536044,27.255358227],[0.692516726,0.060687774,-0.040025666,0.717729422],[0,0,0,0],[9E+09,9E+09,9E+09,9E+09,9E+09,9E+09]];
    CONST robtarget Target_2190:=[[189.842225393,137.460536498,27.261566098],[0.692516726,0.060687774,-0.040025667,0.717729422],[0,0,0,0],[9E+09,9E+09,9E+09,9E+09,9E+09,9E+09]];
    CONST robtarget Target_2200:=[[189.624230729,137.71376379,27.26801408],[0.692516726,0.060687774,-0.040025667,0.717729422],[0,0,0,0],[9E+09,9E+09,9E+09,9E+09,9E+09,9E+09]];
    CONST robtarget Target_2210:=[[189.395428805,137.947217916,27.274702194],[0.692516726,0.060687774,-0.040025666,0.717729422],[0,0,0,0],[9E+09,9E+09,9E+09,9E+09,9E+09,9E+09]];
    CONST robtarget Target_2220:=[[189.15581962,138.16089888,27.281630408],[0.692516726,0.060687774,-0.040025667,0.717729422],[0,0,0,0],[9E+09,9E+09,9E+09,9E+09,9E+09,9E+09]];
    CONST robtarget Target_2230:=[[188.905403174,138.35480668,27.288798755],[0.692516726,0.060687774,-0.040025667,0.717729422],[0,0,0,0],[9E+09,9E+09,9E+09,9E+09,9E+09,9E+09]];
    CONST robtarget Target_2240:=[[188.644179467,138.528941317,27.296207223],[0.692516726,0.060687774,-0.040025667,0.717729422],[0,0,0,0],[9E+09,9E+09,9E+09,9E+09,9E+09,9E+09]];
    CONST robtarget Target_2250:=[[188.3721485,138.683302789,27.303855813],[0.692516726,0.060687774,-0.040025667,0.717729422],[0,0,0,0],[9E+09,9E+09,9E+09,9E+09,9E+09,9E+09]];
    CONST robtarget Target_2260:=[[188.089310272,138.817891097,27.311744524],[0.692516726,0.060687774,-0.040025667,0.717729422],[0,0,0,0],[9E+09,9E+09,9E+09,9E+09,9E+09,9E+09]];
    CONST robtarget Target_2270:=[[187.795664785,138.932706243,27.319873346],[0.692516726,0.060687774,-0.040025666,0.717729422],[0,0,0,0],[9E+09,9E+09,9E+09,9E+09,9E+09,9E+09]];
    CONST robtarget Target_2280:=[[187.491212036,139.027748225,27.3282423],[0.692516726,0.060687774,-0.040025666,0.717729422],[0,0,0,0],[9E+09,9E+09,9E+09,9E+09,9E+09,9E+09]];
    CONST robtarget Target_2290:=[[187.175952026,139.103017042,27.336851388],[0.692516726,0.060687774,-0.040025667,0.717729422],[0,0,0,0],[9E+09,9E+09,9E+09,9E+09,9E+09,9E+09]];
    CONST robtarget Target_2300:=[[186.849884756,139.158512697,27.345700574],[0.692516726,0.060687774,-0.040025666,0.717729422],[0,0,0,0],[9E+09,9E+09,9E+09,9E+09,9E+09,9E+09]];
    CONST robtarget Target_2310:=[[186.513010225,139.194235185,27.354789904],[0.692516726,0.060687774,-0.040025667,0.717729422],[0,0,0,0],[9E+09,9E+09,9E+09,9E+09,9E+09,9E+09]];
    CONST robtarget Target_2320:=[[186.165328434,139.210184512,27.364119345],[0.692516726,0.060687774,-0.040025667,0.717729422],[0,0,0,0],[9E+09,9E+09,9E+09,9E+09,9E+09,9E+09]];
    CONST robtarget Target_2330:=[[185.806839383,139.206360674,27.373688907],[0.692516726,0.060687774,-0.040025667,0.717729422],[0,0,0,0],[9E+09,9E+09,9E+09,9E+09,9E+09,9E+09]];
    CONST robtarget Target_2340:=[[180.816311169,139.018332069,27.506575167],[0.692516726,0.060687774,-0.040025667,0.717729422],[0,0,0,0],[9E+09,9E+09,9E+09,9E+09,9E+09,9E+09]];
    CONST robtarget Target_2350:=[[180.721712314,141.535274246,27.515295936],[0.692516726,0.060687774,-0.040025667,0.717729422],[0,0,0,0],[9E+09,9E+09,9E+09,9E+09,9E+09,9E+09]];
    CONST robtarget Target_2360:=[[179.920388737,141.609064033,-2.473909382],[0.692516726,0.060687774,-0.040025667,0.717729422],[0,0,0,0],[9E+09,9E+09,9E+09,9E+09,9E+09,9E+09]];
    CONST robtarget Target_2370:=[[172.857554936,130.073585442,-2.313571198],[0.692516726,0.060687774,-0.040025667,0.717729422],[0,0,0,0],[9E+09,9E+09,9E+09,9E+09,9E+09,9E+09]];
    CONST robtarget Target_2380:=[[173.658878513,129.999795655,27.67563412],[0.692516726,0.060687774,-0.040025667,0.717729422],[0,0,0,0],[9E+09,9E+09,9E+09,9E+09,9E+09,9E+09]];
    CONST robtarget Target_2390:=[[173.095194424,144.997442841,27.72759837],[0.692516726,0.060687774,-0.040025667,0.717729422],[0,0,0,0],[9E+09,9E+09,9E+09,9E+09,9E+09,9E+09]];
    CONST robtarget Target_2400:=[[173.064705988,145.289224878,27.729130976],[0.692516726,0.060687774,-0.040025667,0.717729422],[0,0,0,0],[9E+09,9E+09,9E+09,9E+09,9E+09,9E+09]];
    CONST robtarget Target_2410:=[[172.996694942,145.540535739,27.731566609],[0.692516726,0.060687774,-0.040025666,0.717729422],[0,0,0,0],[9E+09,9E+09,9E+09,9E+09,9E+09,9E+09]];
    CONST robtarget Target_2420:=[[172.891161285,145.751375422,27.734905291],[0.692516726,0.060687774,-0.040025666,0.717729422],[0,0,0,0],[9E+09,9E+09,9E+09,9E+09,9E+09,9E+09]];
    CONST robtarget Target_2430:=[[172.748105019,145.921743929,27.739147022],[0.692516726,0.060687774,-0.040025667,0.717729422],[0,0,0,0],[9E+09,9E+09,9E+09,9E+09,9E+09,9E+09]];
    CONST robtarget Target_2440:=[[172.567526141,146.051641261,27.744291769],[0.692516726,0.060687774,-0.040025666,0.717729422],[0,0,0,0],[9E+09,9E+09,9E+09,9E+09,9E+09,9E+09]];
    CONST robtarget Target_2450:=[[172.349424655,146.141067413,27.750339587],[0.692516726,0.060687774,-0.040025666,0.717729422],[0,0,0,0],[9E+09,9E+09,9E+09,9E+09,9E+09,9E+09]];
    CONST robtarget Target_2460:=[[172.093800556,146.190022392,27.757290399],[0.692516726,0.060687774,-0.040025666,0.717729422],[0,0,0,0],[9E+09,9E+09,9E+09,9E+09,9E+09,9E+09]];
    CONST robtarget Target_2470:=[[171.800653847,146.19850619,27.765144283],[0.692516726,0.060687774,-0.040025667,0.717729422],[0,0,0,0],[9E+09,9E+09,9E+09,9E+09,9E+09,9E+09]];
    CONST robtarget Target_2480:=[[165.541699714,145.962686981,27.9318058],[0.692516726,0.060687774,-0.040025667,0.717729422],[0,0,0,0],[9E+09,9E+09,9E+09,9E+09,9E+09,9E+09]];
    CONST robtarget Target_2490:=[[165.027738035,145.920701635,27.945435755],[0.692516726,0.060687774,-0.040025667,0.717729422],[0,0,0,0],[9E+09,9E+09,9E+09,9E+09,9E+09,9E+09]];
    CONST robtarget Target_2500:=[[164.535943311,145.834309947,27.958364137],[0.692516726,0.060687774,-0.040025667,0.717729422],[0,0,0,0],[9E+09,9E+09,9E+09,9E+09,9E+09,9E+09]];
    CONST robtarget Target_2510:=[[164.06631554,145.703511918,27.970590944],[0.692516726,0.060687774,-0.040025667,0.717729422],[0,0,0,0],[9E+09,9E+09,9E+09,9E+09,9E+09,9E+09]];
    CONST robtarget Target_2520:=[[163.618854725,145.52830755,27.982116178],[0.692516726,0.060687774,-0.040025667,0.717729422],[0,0,0,0],[9E+09,9E+09,9E+09,9E+09,9E+09,9E+09]];
    CONST robtarget Target_2530:=[[163.193560862,145.308696839,27.992939838],[0.692516726,0.060687774,-0.040025667,0.717729422],[0,0,0,0],[9E+09,9E+09,9E+09,9E+09,9E+09,9E+09]];
    CONST robtarget Target_2540:=[[162.790433955,145.044679789,28.003061914],[0.692516726,0.060687774,-0.040025666,0.717729422],[0,0,0,0],[9E+09,9E+09,9E+09,9E+09,9E+09,9E+09]];
    CONST robtarget Target_2550:=[[162.409474002,144.736256397,28.012482427],[0.692516726,0.060687774,-0.040025666,0.717729422],[0,0,0,0],[9E+09,9E+09,9E+09,9E+09,9E+09,9E+09]];
    CONST robtarget Target_2560:=[[162.050681002,144.383426664,28.021201366],[0.692516726,0.060687774,-0.040025666,0.717729422],[0,0,0,0],[9E+09,9E+09,9E+09,9E+09,9E+09,9E+09]];
    CONST robtarget Target_2570:=[[161.725937117,143.999006462,28.02893277],[0.692516726,0.060687774,-0.040025666,0.717729422],[0,0,0,0],[9E+09,9E+09,9E+09,9E+09,9E+09,9E+09]];
    CONST robtarget Target_2580:=[[161.447124506,143.595811664,28.035390686],[0.692516726,0.060687774,-0.040025667,0.717729422],[0,0,0,0],[9E+09,9E+09,9E+09,9E+09,9E+09,9E+09]];
    CONST robtarget Target_2590:=[[161.214243169,143.173842272,28.040575083],[0.692516726,0.060687774,-0.040025666,0.717729422],[0,0,0,0],[9E+09,9E+09,9E+09,9E+09,9E+09,9E+09]];
    CONST robtarget Target_2600:=[[161.027293106,142.733098284,28.044485994],[0.692516726,0.060687774,-0.040025666,0.717729422],[0,0,0,0],[9E+09,9E+09,9E+09,9E+09,9E+09,9E+09]];
    CONST robtarget Target_2610:=[[160.886274316,142.2735797,28.047123406],[0.692516726,0.060687774,-0.040025666,0.717729422],[0,0,0,0],[9E+09,9E+09,9E+09,9E+09,9E+09,9E+09]];
    CONST robtarget Target_2620:=[[160.791186802,141.795286519,28.048487332],[0.692516726,0.060687774,-0.040025667,0.717729422],[0,0,0,0],[9E+09,9E+09,9E+09,9E+09,9E+09,9E+09]];
    CONST robtarget Target_2630:=[[160.742030561,141.298218745,28.048577737],[0.692516726,0.060687774,-0.040025666,0.717729422],[0,0,0,0],[9E+09,9E+09,9E+09,9E+09,9E+09,9E+09]];
    CONST robtarget Target_2640:=[[160.738805595,140.782376372,28.047394667],[0.692516726,0.060687774,-0.040025667,0.717729422],[0,0,0,0],[9E+09,9E+09,9E+09,9E+09,9E+09,9E+09]];
    CONST robtarget Target_2650:=[[161.161764114,129.528940689,28.008403462],[0.692516726,0.060687774,-0.040025667,0.717729422],[0,0,0,0],[9E+09,9E+09,9E+09,9E+09,9E+09,9E+09]];
    CONST robtarget Target_2660:=[[160.360440537,129.602730476,-1.980801856],[0.692516726,0.060687774,-0.040025667,0.717729422],[0,0,0,0],[9E+09,9E+09,9E+09,9E+09,9E+09,9E+09]];
    CONST robtarget Target_2670:=[[236.945340524,89.071860951,-4.126909086],[0.692516726,0.060687774,-0.040025667,0.717729422],[-2,0,-1,0],[9E+09,9E+09,9E+09,9E+09,9E+09,9E+09]];
    CONST robtarget Target_2680:=[[237.746664101,88.998071164,25.862296232],[0.692516726,0.060687774,-0.040025667,0.717729422],[-2,0,-1,0],[9E+09,9E+09,9E+09,9E+09,9E+09,9E+09]];
    CONST robtarget Target_2690:=[[238.038344918,89.028589567,25.854577496],[0.692516726,0.060687774,-0.040025666,0.717729422],[-2,0,-1,0],[9E+09,9E+09,9E+09,9E+09,9E+09,9E+09]];
    CONST robtarget Target_2700:=[[238.289571342,89.0966412,25.848032069],[0.692516726,0.060687774,-0.040025667,0.717729422],[-2,0,-1,0],[9E+09,9E+09,9E+09,9E+09,9E+09,9E+09]];
    CONST robtarget Target_2710:=[[238.500343372,89.202226061,25.842659953],[0.692516726,0.060687774,-0.040025667,0.717729422],[-2,0,-1,0],[9E+09,9E+09,9E+09,9E+09,9E+09,9E+09]];
    CONST robtarget Target_2720:=[[238.67066101,89.345344153,25.838461146],[0.692516726,0.060687774,-0.040025666,0.717729422],[-2,0,-1,0],[9E+09,9E+09,9E+09,9E+09,9E+09,9E+09]];
    CONST robtarget Target_2730:=[[238.800524255,89.525995474,25.835435648],[0.692516726,0.060687774,-0.040025667,0.717729422],[-2,0,-1,0],[9E+09,9E+09,9E+09,9E+09,9E+09,9E+09]];
    CONST robtarget Target_2740:=[[238.889933107,89.744180026,25.833583461],[0.692516726,0.060687774,-0.040025666,0.717729422],[-2,0,-1,0],[9E+09,9E+09,9E+09,9E+09,9E+09,9E+09]];
    CONST robtarget Target_2750:=[[238.938887565,89.999897806,25.832904583],[0.692516726,0.060687774,-0.040025667,0.717729422],[-2,0,-1,0],[9E+09,9E+09,9E+09,9E+09,9E+09,9E+09]];
    CONST robtarget Target_2760:=[[238.947387631,90.293148816,25.833399015],[0.692516726,0.060687774,-0.040025667,0.717729422],[-2,0,-1,0],[9E+09,9E+09,9E+09,9E+09,9E+09,9E+09]];
    CONST robtarget Target_2770:=[[238.102252402,112.779219009,25.911309354],[0.692516726,0.060687774,-0.040025667,0.717729422],[-2,0,-1,0],[9E+09,9E+09,9E+09,9E+09,9E+09,9E+09]];
    CONST robtarget Target_2780:=[[238.071763965,113.071001045,25.91284196],[0.692516726,0.060687774,-0.040025667,0.717729422],[-2,0,-1,0],[9E+09,9E+09,9E+09,9E+09,9E+09,9E+09]];
    CONST robtarget Target_2790:=[[238.00375292,113.322311906,25.915277604],[0.692516726,0.060687774,-0.040025666,0.717729422],[-2,0,-1,0],[9E+09,9E+09,9E+09,9E+09,9E+09,9E+09]];
    CONST robtarget Target_2800:=[[237.898219262,113.53315159,25.918616286],[0.692516726,0.060687774,-0.040025666,0.717729422],[-2,0,-1,0],[9E+09,9E+09,9E+09,9E+09,9E+09,9E+09]];
    CONST robtarget Target_2810:=[[237.755162996,113.703520097,25.922858006],[0.692516726,0.060687774,-0.040025667,0.717729422],[-2,0,-1,0],[9E+09,9E+09,9E+09,9E+09,9E+09,9E+09]];
    CONST robtarget Target_2820:=[[237.574584119,113.833417427,25.928002764],[0.692516726,0.060687774,-0.040025666,0.717729422],[-2,0,-1,0],[9E+09,9E+09,9E+09,9E+09,9E+09,9E+09]];
    CONST robtarget Target_2830:=[[237.356482632,113.922843581,25.93405056],[0.692516726,0.060687774,-0.040025666,0.717729422],[-2,0,-1,0],[9E+09,9E+09,9E+09,9E+09,9E+09,9E+09]];
    CONST robtarget Target_2840:=[[237.100858533,113.971798558,25.941001394],[0.692516726,0.060687774,-0.040025666,0.717729422],[-2,0,-1,0],[9E+09,9E+09,9E+09,9E+09,9E+09,9E+09]];
    CONST robtarget Target_2850:=[[236.807711825,113.980282358,25.948855267],[0.692516726,0.060687774,-0.040025667,0.717729422],[-2,0,-1,0],[9E+09,9E+09,9E+09,9E+09,9E+09,9E+09]];
    CONST robtarget Target_2860:=[[236.640752645,113.964227463,25.953276979],[0.692516726,0.060687774,-0.040025667,0.717729422],[-2,0,-1,0],[9E+09,9E+09,9E+09,9E+09,9E+09,9E+09]];
    CONST robtarget Target_2870:=[[236.482973919,113.928989743,25.957406186],[0.692516726,0.060687774,-0.040025667,0.717729422],[-2,0,-1,0],[9E+09,9E+09,9E+09,9E+09,9E+09,9E+09]];
    CONST robtarget Target_2880:=[[236.334375648,113.874569201,25.961242887],[0.692516726,0.060687774,-0.040025666,0.717729422],[-2,0,-1,0],[9E+09,9E+09,9E+09,9E+09,9E+09,9E+09]];
    CONST robtarget Target_2890:=[[236.194957831,113.800965833,25.964787082],[0.692516726,0.060687774,-0.040025666,0.717729422],[-2,0,-1,0],[9E+09,9E+09,9E+09,9E+09,9E+09,9E+09]];
    CONST robtarget Target_2900:=[[236.064720468,113.708179643,25.968038772],[0.692516726,0.060687774,-0.040025667,0.717729422],[-2,0,-1,0],[9E+09,9E+09,9E+09,9E+09,9E+09,9E+09]];
    CONST robtarget Target_2910:=[[235.94366356,113.596210627,25.970997957],[0.692516726,0.060687774,-0.040025667,0.717729422],[-2,0,-1,0],[9E+09,9E+09,9E+09,9E+09,9E+09,9E+09]];
    CONST robtarget Target_2920:=[[235.831787106,113.465058787,25.973664635],[0.692516726,0.060687774,-0.040025666,0.717729422],[-2,0,-1,0],[9E+09,9E+09,9E+09,9E+09,9E+09,9E+09]];
    CONST robtarget Target_2930:=[[235.729091106,113.314724124,25.976038808],[0.692516726,0.060687774,-0.040025666,0.717729422],[-2,0,-1,0],[9E+09,9E+09,9E+09,9E+09,9E+09,9E+09]];
    CONST robtarget Target_2940:=[[229.684993721,103.484079065,26.113350767],[0.692516726,0.060687774,-0.040025667,0.717729422],[-1,-1,0,0],[9E+09,9E+09,9E+09,9E+09,9E+09,9E+09]];
    CONST robtarget Target_2950:=[[222.896147591,112.914538618,26.317955524],[0.692516726,0.060687774,-0.040025667,0.717729422],[-1,-1,0,0],[9E+09,9E+09,9E+09,9E+09,9E+09,9E+09]];
    CONST robtarget Target_2960:=[[222.797486135,113.037758001,26.320894985],[0.692516726,0.060687774,-0.040025666,0.717729422],[-1,-1,0,0],[9E+09,9E+09,9E+09,9E+09,9E+09,9E+09]];
    CONST robtarget Target_2970:=[[222.688413158,113.143660219,26.324070036],[0.692516726,0.060687774,-0.040025666,0.717729422],[-1,-1,0,0],[9E+09,9E+09,9E+09,9E+09,9E+09,9E+09]];
    CONST robtarget Target_2980:=[[222.568928658,113.232245274,26.327480677],[0.692516726,0.060687774,-0.040025667,0.717729422],[-1,-1,0,0],[9E+09,9E+09,9E+09,9E+09,9E+09,9E+09]];
    CONST robtarget Target_2990:=[[222.439032635,113.303513165,26.331126908],[0.692516726,0.060687774,-0.040025667,0.717729422],[-1,-1,0,0],[9E+09,9E+09,9E+09,9E+09,9E+09,9E+09]];
    CONST robtarget Target_3000:=[[222.29872509,113.357463892,26.33500873],[0.692516726,0.060687774,-0.040025667,0.717729422],[-1,-1,0,0],[9E+09,9E+09,9E+09,9E+09,9E+09,9E+09]];
    CONST robtarget Target_3010:=[[222.148006022,113.394097455,26.339126143],[0.692516726,0.060687774,-0.040025666,0.717729422],[-1,-1,0,0],[9E+09,9E+09,9E+09,9E+09,9E+09,9E+09]];
    CONST robtarget Target_3020:=[[221.986875432,113.413413855,26.343479145],[0.692516726,0.060687774,-0.040025666,0.717729422],[-1,-1,0,0],[9E+09,9E+09,9E+09,9E+09,9E+09,9E+09]];
    CONST robtarget Target_3030:=[[221.815333319,113.415413089,26.348067739],[0.692516726,0.060687774,-0.040025667,0.717729422],[-1,-1,0,0],[9E+09,9E+09,9E+09,9E+09,9E+09,9E+09]];
    CONST robtarget Target_3040:=[[221.523652502,113.384894687,26.355786475],[0.692516726,0.060687774,-0.040025666,0.717729422],[-1,-1,0,0],[9E+09,9E+09,9E+09,9E+09,9E+09,9E+09]];
    CONST robtarget Target_3050:=[[221.272426078,113.316843054,26.362331902],[0.692516726,0.060687774,-0.040025667,0.717729422],[-1,-1,0,0],[9E+09,9E+09,9E+09,9E+09,9E+09,9E+09]];
    CONST robtarget Target_3060:=[[221.061654048,113.211258193,26.367704018],[0.692516726,0.060687774,-0.040025667,0.717729422],[-1,-1,0,0],[9E+09,9E+09,9E+09,9E+09,9E+09,9E+09]];
    CONST robtarget Target_3070:=[[220.89133641,113.068140101,26.371902825],[0.692516726,0.060687774,-0.040025666,0.717729422],[-1,-1,0,0],[9E+09,9E+09,9E+09,9E+09,9E+09,9E+09]];
    CONST robtarget Target_3080:=[[220.761473165,112.88748878,26.374928323],[0.692516726,0.060687774,-0.040025667,0.717729422],[-1,-1,0,0],[9E+09,9E+09,9E+09,9E+09,9E+09,9E+09]];
    CONST robtarget Target_3090:=[[220.672064313,112.669304229,26.37678051],[0.692516726,0.060687774,-0.040025666,0.717729422],[-1,-1,0,0],[9E+09,9E+09,9E+09,9E+09,9E+09,9E+09]];
    CONST robtarget Target_3100:=[[220.623109854,112.413586447,26.377459388],[0.692516726,0.060687774,-0.040025667,0.717729422],[-1,-1,0,0],[9E+09,9E+09,9E+09,9E+09,9E+09,9E+09]];
    CONST robtarget Target_3110:=[[220.614609789,112.120335438,26.376964955],[0.692516726,0.060687774,-0.040025667,0.717729422],[-1,-1,0,0],[9E+09,9E+09,9E+09,9E+09,9E+09,9E+09]];
    CONST robtarget Target_3120:=[[221.459745018,89.634265245,26.299054617],[0.692516726,0.060687774,-0.040025667,0.717729422],[-1,-1,0,0],[9E+09,9E+09,9E+09,9E+09,9E+09,9E+09]];
    CONST robtarget Target_3130:=[[220.658421441,89.708055033,-3.690150701],[0.692516726,0.060687774,-0.040025667,0.717729422],[-1,-1,0,0],[9E+09,9E+09,9E+09,9E+09,9E+09,9E+09]];
    CONST robtarget Target_3140:=[[215.291843232,99.52539161,-3.522597584],[0.692516726,0.060687774,-0.040025667,0.717729422],[0,0,0,0],[9E+09,9E+09,9E+09,9E+09,9E+09,9E+09]];
    CONST robtarget Target_3150:=[[216.093166809,99.451601822,26.466607734],[0.692516726,0.060687774,-0.040025667,0.717729422],[0,0,0,0],[9E+09,9E+09,9E+09,9E+09,9E+09,9E+09]];
    CONST robtarget Target_3160:=[[216.040778939,100.08366034,26.469562767],[0.692516726,0.060687774,-0.040025667,0.717729422],[0,0,0,0],[9E+09,9E+09,9E+09,9E+09,9E+09,9E+09]];
    CONST robtarget Target_3170:=[[215.932087467,100.690163041,26.473959374],[0.692516726,0.060687774,-0.040025666,0.717729422],[0,0,0,0],[9E+09,9E+09,9E+09,9E+09,9E+09,9E+09]];
    CONST robtarget Target_3180:=[[215.767092394,101.271109926,26.479797555],[0.692516726,0.060687774,-0.040025666,0.717729422],[0,0,0,0],[9E+09,9E+09,9E+09,9E+09,9E+09,9E+09]];
    CONST robtarget Target_3190:=[[215.54579372,101.826500994,26.487077309],[0.692516726,0.060687774,-0.040025666,0.717729422],[0,0,0,0],[9E+09,9E+09,9E+09,9E+09,9E+09,9E+09]];
    CONST robtarget Target_3200:=[[215.268191445,102.356336246,26.495798636],[0.692516726,0.060687774,-0.040025666,0.717729422],[0,0,0,0],[9E+09,9E+09,9E+09,9E+09,9E+09,9E+09]];
    CONST robtarget Target_3210:=[[214.93428557,102.860615682,26.505961537],[0.692516726,0.060687774,-0.040025667,0.717729422],[0,0,0,0],[9E+09,9E+09,9E+09,9E+09,9E+09,9E+09]];
    CONST robtarget Target_3220:=[[214.544076093,103.339339301,26.517566011],[0.692516726,0.060687774,-0.040025666,0.717729422],[0,0,0,0],[9E+09,9E+09,9E+09,9E+09,9E+09,9E+09]];
    CONST robtarget Target_3230:=[[214.097563016,103.792507104,26.530612059],[0.692516726,0.060687774,-0.040025667,0.717729422],[0,0,0,0],[9E+09,9E+09,9E+09,9E+09,9E+09,9E+09]];
    CONST robtarget Target_3240:=[[213.611951669,104.20384245,26.544599898],[0.692516726,0.060687774,-0.040025667,0.717729422],[0,0,0,0],[9E+09,9E+09,9E+09,9E+09,9E+09,9E+09]];
    CONST robtarget Target_3250:=[[213.104447389,104.557068697,26.559029745],[0.692516726,0.060687774,-0.040025667,0.717729422],[0,0,0,0],[9E+09,9E+09,9E+09,9E+09,9E+09,9E+09]];
    CONST robtarget Target_3260:=[[212.575050172,104.852185846,26.5739016],[0.692516726,0.060687774,-0.040025667,0.717729422],[0,0,0,0],[9E+09,9E+09,9E+09,9E+09,9E+09,9E+09]];
    CONST robtarget Target_3270:=[[212.02376002,105.089193898,26.589215462],[0.692516726,0.060687774,-0.040025666,0.717729422],[0,0,0,0],[9E+09,9E+09,9E+09,9E+09,9E+09,9E+09]];
    CONST robtarget Target_3280:=[[211.450576933,105.26809285,26.604971333],[0.692516726,0.060687774,-0.040025667,0.717729422],[0,0,0,0],[9E+09,9E+09,9E+09,9E+09,9E+09,9E+09]];
    CONST robtarget Target_3290:=[[210.85550091,105.388882704,26.621169211],[0.692516726,0.060687774,-0.040025667,0.717729422],[0,0,0,0],[9E+09,9E+09,9E+09,9E+09,9E+09,9E+09]];
    CONST robtarget Target_3300:=[[210.238531953,105.451563461,26.637809098],[0.692516726,0.060687774,-0.040025666,0.717729422],[0,0,0,0],[9E+09,9E+09,9E+09,9E+09,9E+09,9E+09]];
    CONST robtarget Target_3310:=[[209.599670059,105.456135118,26.654890992],[0.692516726,0.060687774,-0.040025667,0.717729422],[0,0,0,0],[9E+09,9E+09,9E+09,9E+09,9E+09,9E+09]];
    CONST robtarget Target_3320:=[[208.958397265,105.403657183,26.671896934],[0.692516726,0.060687774,-0.040025666,0.717729422],[0,0,0,0],[9E+09,9E+09,9E+09,9E+09,9E+09,9E+09]];
    CONST robtarget Target_3330:=[[208.34459254,105.295580886,26.688032115],[0.692516726,0.060687774,-0.040025667,0.717729422],[0,0,0,0],[9E+09,9E+09,9E+09,9E+09,9E+09,9E+09]];
    CONST robtarget Target_3340:=[[207.758255883,105.131906226,26.703296537],[0.692516726,0.060687774,-0.040025666,0.717729422],[0,0,0,0],[9E+09,9E+09,9E+09,9E+09,9E+09,9E+09]];
    CONST robtarget Target_3350:=[[207.199387296,104.912633206,26.717690198],[0.692516726,0.060687774,-0.040025666,0.717729422],[0,0,0,0],[9E+09,9E+09,9E+09,9E+09,9E+09,9E+09]];
    CONST robtarget Target_3360:=[[206.667986776,104.637761823,26.731213099],[0.692516726,0.060687774,-0.040025667,0.717729422],[0,0,0,0],[9E+09,9E+09,9E+09,9E+09,9E+09,9E+09]];
    CONST robtarget Target_3370:=[[206.164054325,104.307292078,26.743865241],[0.692516726,0.060687774,-0.040025667,0.717729422],[0,0,0,0],[9E+09,9E+09,9E+09,9E+09,9E+09,9E+09]];
    CONST robtarget Target_3380:=[[205.687589943,103.921223973,26.755646622],[0.692516726,0.060687774,-0.040025666,0.717729422],[0,0,0,0],[9E+09,9E+09,9E+09,9E+09,9E+09,9E+09]];
    CONST robtarget Target_3390:=[[205.238593629,103.479557505,26.766557243],[0.692516726,0.060687774,-0.040025666,0.717729422],[0,0,0,0],[9E+09,9E+09,9E+09,9E+09,9E+09,9E+09]];
    CONST robtarget Target_3400:=[[204.832074428,102.998481145,26.776235889],[0.692516726,0.060687774,-0.040025667,0.717729422],[0,0,0,0],[9E+09,9E+09,9E+09,9E+09,9E+09,9E+09]];
    CONST robtarget Target_3410:=[[204.483041383,102.494183365,26.784321344],[0.692516726,0.060687774,-0.040025667,0.717729422],[0,0,0,0],[9E+09,9E+09,9E+09,9E+09,9E+09,9E+09]];
    CONST robtarget Target_3420:=[[204.191494495,101.966664165,26.790813609],[0.692516726,0.060687774,-0.040025666,0.717729422],[0,0,0,0],[9E+09,9E+09,9E+09,9E+09,9E+09,9E+09]];
    CONST robtarget Target_3430:=[[203.957433765,101.415923544,26.795712683],[0.692516726,0.060687774,-0.040025666,0.717729422],[0,0,0,0],[9E+09,9E+09,9E+09,9E+09,9E+09,9E+09]];
    CONST robtarget Target_3440:=[[203.780859191,100.841961503,26.799018567],[0.692516726,0.060687774,-0.040025667,0.717729422],[0,0,0,0],[9E+09,9E+09,9E+09,9E+09,9E+09,9E+09]];
    CONST robtarget Target_3450:=[[203.661770773,100.244778041,26.800731261],[0.692516726,0.060687774,-0.040025667,0.717729422],[0,0,0,0],[9E+09,9E+09,9E+09,9E+09,9E+09,9E+09]];
    CONST robtarget Target_3460:=[[203.600168513,99.62437316,26.800850764],[0.692516726,0.060687774,-0.040025667,0.717729422],[0,0,0,0],[9E+09,9E+09,9E+09,9E+09,9E+09,9E+09]];
    CONST robtarget Target_3470:=[[203.59605241,98.980746856,26.799377076],[0.692516726,0.060687774,-0.040025667,0.717729422],[0,0,0,0],[9E+09,9E+09,9E+09,9E+09,9E+09,9E+09]];
    CONST robtarget Target_3480:=[[203.784468312,93.967663678,26.782007611],[0.692516726,0.060687774,-0.040025667,0.717729422],[0,0,0,0],[9E+09,9E+09,9E+09,9E+09,9E+09,9E+09]];
    CONST robtarget Target_3490:=[[203.836856183,93.33560516,26.779052578],[0.692516726,0.060687774,-0.040025667,0.717729422],[0,0,0,0],[9E+09,9E+09,9E+09,9E+09,9E+09,9E+09]];
    CONST robtarget Target_3500:=[[203.945547655,92.72910246,26.774655971],[0.692516726,0.060687774,-0.040025666,0.717729422],[0,0,0,0],[9E+09,9E+09,9E+09,9E+09,9E+09,9E+09]];
    CONST robtarget Target_3510:=[[204.110542727,92.148155574,26.768817791],[0.692516726,0.060687774,-0.040025666,0.717729422],[0,0,0,0],[9E+09,9E+09,9E+09,9E+09,9E+09,9E+09]];
    CONST robtarget Target_3520:=[[204.331841401,91.592764506,26.761538037],[0.692516726,0.060687774,-0.040025666,0.717729422],[0,0,0,0],[9E+09,9E+09,9E+09,9E+09,9E+09,9E+09]];
    CONST robtarget Target_3530:=[[204.609443676,91.062929254,26.75281671],[0.692516726,0.060687774,-0.040025666,0.717729422],[0,0,0,0],[9E+09,9E+09,9E+09,9E+09,9E+09,9E+09]];
    CONST robtarget Target_3540:=[[204.943349551,90.558649819,26.742653809],[0.692516726,0.060687774,-0.040025667,0.717729422],[0,0,0,0],[9E+09,9E+09,9E+09,9E+09,9E+09,9E+09]];
    CONST robtarget Target_3550:=[[205.333559028,90.0799262,26.731049334],[0.692516726,0.060687774,-0.040025666,0.717729422],[0,0,0,0],[9E+09,9E+09,9E+09,9E+09,9E+09,9E+09]];
    CONST robtarget Target_3560:=[[205.780072106,89.626758396,26.718003286],[0.692516726,0.060687774,-0.040025667,0.717729422],[0,0,0,0],[9E+09,9E+09,9E+09,9E+09,9E+09,9E+09]];
    CONST robtarget Target_3570:=[[206.265358547,89.215410809,26.704024099],[0.692516726,0.060687774,-0.040025667,0.717729422],[0,0,0,0],[9E+09,9E+09,9E+09,9E+09,9E+09,9E+09]];
    CONST robtarget Target_3580:=[[206.771888115,88.862147837,26.689620207],[0.692516726,0.060687774,-0.040025667,0.717729422],[0,0,0,0],[9E+09,9E+09,9E+09,9E+09,9E+09,9E+09]];
    CONST robtarget Target_3590:=[[207.299660812,88.566969481,26.674791609],[0.692516726,0.060687774,-0.040025667,0.717729422],[0,0,0,0],[9E+09,9E+09,9E+09,9E+09,9E+09,9E+09]];
    CONST robtarget Target_3600:=[[207.848676634,88.329875739,26.659538307],[0.692516726,0.060687774,-0.040025666,0.717729422],[0,0,0,0],[9E+09,9E+09,9E+09,9E+09,9E+09,9E+09]];
    CONST robtarget Target_3610:=[[208.418935584,88.150866615,26.643860299],[0.692516726,0.060687774,-0.040025667,0.717729422],[0,0,0,0],[9E+09,9E+09,9E+09,9E+09,9E+09,9E+09]];
    CONST robtarget Target_3620:=[[209.01043766,88.029942104,26.627757587],[0.692516726,0.060687774,-0.040025666,0.717729422],[0,0,0,0],[9E+09,9E+09,9E+09,9E+09,9E+09,9E+09]];
    CONST robtarget Target_3630:=[[209.623182864,87.967102209,26.611230169],[0.692516726,0.060687774,-0.040025667,0.717729422],[0,0,0,0],[9E+09,9E+09,9E+09,9E+09,9E+09,9E+09]];
    CONST robtarget Target_3640:=[[210.257171194,87.962346929,26.594278046],[0.692516726,0.060687774,-0.040025667,0.717729422],[0,0,0,0],[9E+09,9E+09,9E+09,9E+09,9E+09,9E+09]];
    CONST robtarget Target_3650:=[[210.893883114,88.014978503,26.577394351],[0.692516726,0.060687774,-0.040025667,0.717729422],[0,0,0,0],[9E+09,9E+09,9E+09,9E+09,9E+09,9E+09]];
    CONST robtarget Target_3660:=[[211.50440215,88.123907441,26.561349062],[0.692516726,0.060687774,-0.040025667,0.717729422],[0,0,0,0],[9E+09,9E+09,9E+09,9E+09,9E+09,9E+09]];
    CONST robtarget Target_3670:=[[212.088728303,88.289133743,26.54614218],[0.692516726,0.060687774,-0.040025667,0.717729422],[0,0,0,0],[9E+09,9E+09,9E+09,9E+09,9E+09,9E+09]];
    CONST robtarget Target_3680:=[[212.646861572,88.510657409,26.531773705],[0.692516726,0.060687774,-0.040025666,0.717729422],[0,0,0,0],[9E+09,9E+09,9E+09,9E+09,9E+09,9E+09]];
    CONST robtarget Target_3690:=[[213.178801958,88.788478441,26.518243636],[0.692516726,0.060687774,-0.040025667,0.717729422],[0,0,0,0],[9E+09,9E+09,9E+09,9E+09,9E+09,9E+09]];
    CONST robtarget Target_3700:=[[213.684549461,89.122596835,26.505551973],[0.692516726,0.060687774,-0.040025667,0.717729422],[0,0,0,0],[9E+09,9E+09,9E+09,9E+09,9E+09,9E+09]];
    CONST robtarget Target_3710:=[[214.16410408,89.513012595,26.493698717],[0.692516726,0.060687774,-0.040025666,0.717729422],[0,0,0,0],[9E+09,9E+09,9E+09,9E+09,9E+09,9E+09]];
    CONST robtarget Target_3720:=[[214.617465816,89.959725718,26.482683868],[0.692516726,0.060687774,-0.040025666,0.717729422],[0,0,0,0],[9E+09,9E+09,9E+09,9E+09,9E+09,9E+09]];
    CONST robtarget Target_3730:=[[215.028699775,90.445210938,26.47289009],[0.692516726,0.060687774,-0.040025667,0.717729422],[0,0,0,0],[9E+09,9E+09,9E+09,9E+09,9E+09,9E+09]];
    CONST robtarget Target_3740:=[[215.381871064,90.951942985,26.464700049],[0.692516726,0.060687774,-0.040025667,0.717729422],[0,0,0,0],[9E+09,9E+09,9E+09,9E+09,9E+09,9E+09]];
    CONST robtarget Target_3750:=[[215.676979681,91.479921859,26.458113744],[0.692516726,0.060687774,-0.040025666,0.717729422],[0,0,0,0],[9E+09,9E+09,9E+09,9E+09,9E+09,9E+09]];
    CONST robtarget Target_3760:=[[215.914025628,92.029147561,26.453131176],[0.692516726,0.060687774,-0.040025667,0.717729422],[0,0,0,0],[9E+09,9E+09,9E+09,9E+09,9E+09,9E+09]];
    CONST robtarget Target_3770:=[[216.093008905,92.59962009,26.449752344],[0.692516726,0.060687774,-0.040025667,0.717729422],[0,0,0,0],[9E+09,9E+09,9E+09,9E+09,9E+09,9E+09]];
    CONST robtarget Target_3780:=[[216.213929512,93.191339448,26.447977249],[0.692516726,0.060687774,-0.040025667,0.717729422],[0,0,0,0],[9E+09,9E+09,9E+09,9E+09,9E+09,9E+09]];
    CONST robtarget Target_3790:=[[216.276787447,93.804305632,26.447805891],[0.692516726,0.060687774,-0.040025666,0.717729422],[0,0,0,0],[9E+09,9E+09,9E+09,9E+09,9E+09,9E+09]];
    CONST robtarget Target_3800:=[[216.281582711,94.438518644,26.449238269],[0.692516726,0.060687774,-0.040025667,0.717729422],[0,0,0,0],[9E+09,9E+09,9E+09,9E+09,9E+09,9E+09]];
    CONST robtarget Target_3810:=[[216.093166809,99.451601822,26.466607734],[0.692516726,0.060687774,-0.040025667,0.717729422],[0,0,0,0],[9E+09,9E+09,9E+09,9E+09,9E+09,9E+09]];
    CONST robtarget Target_3820:=[[215.291843232,99.52539161,-3.522597584],[0.692516726,0.060687774,-0.040025667,0.717729422],[0,0,0,0],[9E+09,9E+09,9E+09,9E+09,9E+09,9E+09]];
    CONST robtarget Target_3830:=[[198.193606008,88.859913026,-2.59178875],[0.692516726,0.060687774,-0.040025667,0.717729422],[0,0,0,0],[9E+09,9E+09,9E+09,9E+09,9E+09,9E+09]];
    CONST robtarget Target_3840:=[[198.994929585,88.786123238,27.397416567],[0.692516726,0.060687774,-0.040025667,0.717729422],[0,0,0,0],[9E+09,9E+09,9E+09,9E+09,9E+09,9E+09]];
    CONST robtarget Target_3850:=[[198.431245496,103.783770425,27.449380817],[0.692516726,0.060687774,-0.040025667,0.717729422],[0,0,0,0],[9E+09,9E+09,9E+09,9E+09,9E+09,9E+09]];
    CONST robtarget Target_3860:=[[198.384834518,104.152868157,27.451529119],[0.692516726,0.060687774,-0.040025667,0.717729422],[0,0,0,0],[9E+09,9E+09,9E+09,9E+09,9E+09,9E+09]];
    CONST robtarget Target_3870:=[[198.339930373,104.307231013,27.453108792],[0.692516726,0.060687774,-0.040025667,0.717729422],[0,0,0,0],[9E+09,9E+09,9E+09,9E+09,9E+09,9E+09]];
    CONST robtarget Target_3880:=[[198.275881868,104.454509626,27.455182579],[0.692516726,0.060687774,-0.040025666,0.717729422],[0,0,0,0],[9E+09,9E+09,9E+09,9E+09,9E+09,9E+09]];
    CONST robtarget Target_3890:=[[198.181346008,104.602018746,27.458071568],[0.692516726,0.060687774,-0.040025666,0.717729422],[0,0,0,0],[9E+09,9E+09,9E+09,9E+09,9E+09,9E+09]];
    CONST robtarget Target_3900:=[[198.060849948,104.728938941,27.461603564],[0.692516726,0.060687774,-0.040025667,0.717729422],[0,0,0,0],[9E+09,9E+09,9E+09,9E+09,9E+09,9E+09]];
    CONST robtarget Target_3910:=[[197.902742874,104.838427008,27.466097649],[0.692516726,0.060687774,-0.040025666,0.717729422],[0,0,0,0],[9E+09,9E+09,9E+09,9E+09,9E+09,9E+09]];
    CONST robtarget Target_3920:=[[197.725883977,104.914821881,27.471011362],[0.692516726,0.060687774,-0.040025667,0.717729422],[0,0,0,0],[9E+09,9E+09,9E+09,9E+09,9E+09,9E+09]];
    CONST robtarget Target_3930:=[[197.434874532,104.975809743,27.478937315],[0.692516726,0.060687774,-0.040025666,0.717729422],[0,0,0,0],[9E+09,9E+09,9E+09,9E+09,9E+09,9E+09]];
    CONST robtarget Target_3940:=[[197.13670492,104.984833774,27.48692673],[0.692516726,0.060687774,-0.040025667,0.717729422],[0,0,0,0],[9E+09,9E+09,9E+09,9E+09,9E+09,9E+09]];
    CONST robtarget Target_3950:=[[189.6509126,104.702790866,27.68625612],[0.692516726,0.060687774,-0.040025667,0.717729422],[0,0,0,0],[9E+09,9E+09,9E+09,9E+09,9E+09,9E+09]];
    CONST robtarget Target_3960:=[[189.281942395,104.656339205,27.696000855],[0.692516726,0.060687774,-0.040025666,0.717729422],[0,0,0,0],[9E+09,9E+09,9E+09,9E+09,9E+09,9E+09]];
    CONST robtarget Target_3970:=[[189.127631197,104.611409024,27.700013559],[0.692516726,0.060687774,-0.040025666,0.717729422],[0,0,0,0],[9E+09,9E+09,9E+09,9E+09,9E+09,9E+09]];
    CONST robtarget Target_3980:=[[188.980400475,104.547328173,27.703789949],[0.692516726,0.060687774,-0.040025667,0.717729422],[0,0,0,0],[9E+09,9E+09,9E+09,9E+09,9E+09,9E+09]];
    CONST robtarget Target_3990:=[[188.832937327,104.452749161,27.707497508],[0.692516726,0.060687774,-0.040025666,0.717729422],[0,0,0,0],[9E+09,9E+09,9E+09,9E+09,9E+09,9E+09]];
    CONST robtarget Target_4000:=[[188.706054113,104.332202116,27.710591267],[0.692516726,0.060687774,-0.040025666,0.717729422],[0,0,0,0],[9E+09,9E+09,9E+09,9E+09,9E+09,9E+09]];
    CONST robtarget Target_4010:=[[188.596594389,104.174031892,27.713126889],[0.692516726,0.060687774,-0.040025667,0.717729422],[0,0,0,0],[9E+09,9E+09,9E+09,9E+09,9E+09,9E+09]];
    CONST robtarget Target_4020:=[[188.520214919,103.997105384,27.714732444],[0.692516726,0.060687774,-0.040025667,0.717729422],[0,0,0,0],[9E+09,9E+09,9E+09,9E+09,9E+09,9E+09]];
    CONST robtarget Target_4030:=[[188.459229506,103.705988942,27.715645693],[0.692516726,0.060687774,-0.040025666,0.717729422],[0,0,0,0],[9E+09,9E+09,9E+09,9E+09,9E+09,9E+09]];
    CONST robtarget Target_4040:=[[188.45018907,103.407713215,27.715153336],[0.692516726,0.060687774,-0.040025667,0.717729422],[0,0,0,0],[9E+09,9E+09,9E+09,9E+09,9E+09,9E+09]];
    CONST robtarget Target_4050:=[[188.544006117,100.911572212,27.70650464],[0.692516726,0.060687774,-0.040025667,0.717729422],[0,0,0,0],[9E+09,9E+09,9E+09,9E+09,9E+09,9E+09]];
    CONST robtarget Target_4060:=[[188.590417096,100.542474482,27.704356339],[0.692516726,0.060687774,-0.040025667,0.717729422],[0,0,0,0],[9E+09,9E+09,9E+09,9E+09,9E+09,9E+09]];
    CONST robtarget Target_4070:=[[188.63532124,100.388111626,27.702776665],[0.692516726,0.060687774,-0.040025667,0.717729422],[0,0,0,0],[9E+09,9E+09,9E+09,9E+09,9E+09,9E+09]];
    CONST robtarget Target_4080:=[[188.699369745,100.240833011,27.700702878],[0.692516726,0.060687774,-0.040025666,0.717729422],[0,0,0,0],[9E+09,9E+09,9E+09,9E+09,9E+09,9E+09]];
    CONST robtarget Target_4090:=[[188.793905604,100.093323892,27.697813889],[0.692516726,0.060687774,-0.040025666,0.717729422],[0,0,0,0],[9E+09,9E+09,9E+09,9E+09,9E+09,9E+09]];
    CONST robtarget Target_4100:=[[188.914401665,99.966403697,27.694281893],[0.692516726,0.060687774,-0.040025667,0.717729422],[0,0,0,0],[9E+09,9E+09,9E+09,9E+09,9E+09,9E+09]];
    CONST robtarget Target_4110:=[[189.07250874,99.85691563,27.689787809],[0.692516726,0.060687774,-0.040025666,0.717729422],[0,0,0,0],[9E+09,9E+09,9E+09,9E+09,9E+09,9E+09]];
    CONST robtarget Target_4120:=[[189.249367636,99.780520758,27.684874095],[0.692516726,0.060687774,-0.040025667,0.717729422],[0,0,0,0],[9E+09,9E+09,9E+09,9E+09,9E+09,9E+09]];
    CONST robtarget Target_4130:=[[189.540377081,99.719532894,27.676948143],[0.692516726,0.060687774,-0.040025666,0.717729422],[0,0,0,0],[9E+09,9E+09,9E+09,9E+09,9E+09,9E+09]];
    CONST robtarget Target_4140:=[[189.838546694,99.710508863,27.668958727],[0.692516726,0.060687774,-0.040025667,0.717729422],[0,0,0,0],[9E+09,9E+09,9E+09,9E+09,9E+09,9E+09]];
    CONST robtarget Target_4150:=[[190.207516899,99.756960524,27.659213992],[0.692516726,0.060687774,-0.040025666,0.717729422],[0,0,0,0],[9E+09,9E+09,9E+09,9E+09,9E+09,9E+09]];
    CONST robtarget Target_4160:=[[190.361828097,99.801890706,27.655201288],[0.692516726,0.060687774,-0.040025666,0.717729422],[0,0,0,0],[9E+09,9E+09,9E+09,9E+09,9E+09,9E+09]];
    CONST robtarget Target_4170:=[[190.509058818,99.865971557,27.651424898],[0.692516726,0.060687774,-0.040025667,0.717729422],[0,0,0,0],[9E+09,9E+09,9E+09,9E+09,9E+09,9E+09]];
    CONST robtarget Target_4180:=[[190.656521966,99.960550568,27.647717339],[0.692516726,0.060687774,-0.040025666,0.717729422],[0,0,0,0],[9E+09,9E+09,9E+09,9E+09,9E+09,9E+09]];
    CONST robtarget Target_4190:=[[190.78340518,100.081097613,27.64462358],[0.692516726,0.060687774,-0.040025666,0.717729422],[0,0,0,0],[9E+09,9E+09,9E+09,9E+09,9E+09,9E+09]];
    CONST robtarget Target_4200:=[[190.892864904,100.239267837,27.642087958],[0.692516726,0.060687774,-0.040025667,0.717729422],[0,0,0,0],[9E+09,9E+09,9E+09,9E+09,9E+09,9E+09]];
    CONST robtarget Target_4210:=[[190.969244375,100.416194346,27.640482403],[0.692516726,0.060687774,-0.040025667,0.717729422],[0,0,0,0],[9E+09,9E+09,9E+09,9E+09,9E+09,9E+09]];
    CONST robtarget Target_4220:=[[191.030229788,100.707310787,27.639569154],[0.692516726,0.060687774,-0.040025666,0.717729422],[0,0,0,0],[9E+09,9E+09,9E+09,9E+09,9E+09,9E+09]];
    CONST robtarget Target_4230:=[[191.039270223,101.005586515,27.64006151],[0.692516726,0.060687774,-0.040025667,0.717729422],[0,0,0,0],[9E+09,9E+09,9E+09,9E+09,9E+09,9E+09]];
    CONST robtarget Target_4240:=[[190.9923617,102.253657016,27.644385859],[0.692516726,0.060687774,-0.040025667,0.717729422],[0,0,0,0],[9E+09,9E+09,9E+09,9E+09,9E+09,9E+09]];
    CONST robtarget Target_4250:=[[190.191038123,102.327446804,-2.344819459],[0.692516726,0.060687774,-0.040025667,0.717729422],[0,0,0,0],[9E+09,9E+09,9E+09,9E+09,9E+09,9E+09]];
    CONST robtarget Target_4260:=[[181.355762099,103.24613017,-2.60665686],[0.692516726,0.060687774,-0.040025667,0.717729422],[0,0,0,0],[9E+09,9E+09,9E+09,9E+09,9E+09,9E+09]];
    CONST robtarget Target_4270:=[[182.157085676,103.172340383,27.382548458],[0.692516726,0.060687774,-0.040025667,0.717729422],[0,0,0,0],[9E+09,9E+09,9E+09,9E+09,9E+09,9E+09]];
    CONST robtarget Target_4280:=[[182.12659724,103.464122419,27.384081064],[0.692516726,0.060687774,-0.040025667,0.717729422],[0,0,0,0],[9E+09,9E+09,9E+09,9E+09,9E+09,9E+09]];
    CONST robtarget Target_4290:=[[182.058586193,103.71543328,27.386516708],[0.692516726,0.060687774,-0.040025666,0.717729422],[0,0,0,0],[9E+09,9E+09,9E+09,9E+09,9E+09,9E+09]];
    CONST robtarget Target_4300:=[[181.953052537,103.926272964,27.38985539],[0.692516726,0.060687774,-0.040025666,0.717729422],[0,0,0,0],[9E+09,9E+09,9E+09,9E+09,9E+09,9E+09]];
    CONST robtarget Target_4310:=[[181.80999627,104.09664147,27.39409711],[0.692516726,0.060687774,-0.040025667,0.717729422],[0,0,0,0],[9E+09,9E+09,9E+09,9E+09,9E+09,9E+09]];
    CONST robtarget Target_4320:=[[181.629417392,104.226538801,27.399241868],[0.692516726,0.060687774,-0.040025666,0.717729422],[0,0,0,0],[9E+09,9E+09,9E+09,9E+09,9E+09,9E+09]];
    CONST robtarget Target_4330:=[[181.411315905,104.315964954,27.405289665],[0.692516726,0.060687774,-0.040025666,0.717729422],[0,0,0,0],[9E+09,9E+09,9E+09,9E+09,9E+09,9E+09]];
    CONST robtarget Target_4340:=[[181.155691807,104.364919932,27.412240499],[0.692516726,0.060687774,-0.040025666,0.717729422],[0,0,0,0],[9E+09,9E+09,9E+09,9E+09,9E+09,9E+09]];
    CONST robtarget Target_4350:=[[180.8625451,104.373403732,27.420094371],[0.692516726,0.060687774,-0.040025667,0.717729422],[0,0,0,0],[9E+09,9E+09,9E+09,9E+09,9E+09,9E+09]];
    CONST robtarget Target_4360:=[[175.872016886,104.185375126,27.552980631],[0.692516726,0.060687774,-0.040025667,0.717729422],[0,0,0,0],[9E+09,9E+09,9E+09,9E+09,9E+09,9E+09]];
    CONST robtarget Target_4370:=[[175.358055208,104.14338978,27.566610586],[0.692516726,0.060687774,-0.040025667,0.717729422],[0,0,0,0],[9E+09,9E+09,9E+09,9E+09,9E+09,9E+09]];
    CONST robtarget Target_4380:=[[174.866260483,104.056998092,27.579538967],[0.692516726,0.060687774,-0.040025667,0.717729422],[0,0,0,0],[9E+09,9E+09,9E+09,9E+09,9E+09,9E+09]];
    CONST robtarget Target_4390:=[[174.396632713,103.926200064,27.591765775],[0.692516726,0.060687774,-0.040025667,0.717729422],[0,0,0,0],[9E+09,9E+09,9E+09,9E+09,9E+09,9E+09]];
    CONST robtarget Target_4400:=[[173.949171897,103.750995695,27.603291009],[0.692516726,0.060687774,-0.040025667,0.717729422],[0,0,0,0],[9E+09,9E+09,9E+09,9E+09,9E+09,9E+09]];
    CONST robtarget Target_4410:=[[173.523878035,103.531384984,27.614114669],[0.692516726,0.060687774,-0.040025667,0.717729422],[0,0,0,0],[9E+09,9E+09,9E+09,9E+09,9E+09,9E+09]];
    CONST robtarget Target_4420:=[[173.120751127,103.267367933,27.624236756],[0.692516726,0.060687774,-0.040025666,0.717729422],[0,0,0,0],[9E+09,9E+09,9E+09,9E+09,9E+09,9E+09]];
    CONST robtarget Target_4430:=[[172.739791174,102.958944541,27.633657269],[0.692516726,0.060687774,-0.040025666,0.717729422],[0,0,0,0],[9E+09,9E+09,9E+09,9E+09,9E+09,9E+09]];
    CONST robtarget Target_4440:=[[172.380998174,102.606114808,27.642376208],[0.692516726,0.060687774,-0.040025666,0.717729422],[0,0,0,0],[9E+09,9E+09,9E+09,9E+09,9E+09,9E+09]];
    CONST robtarget Target_4450:=[[172.056254289,102.221694606,27.650107611],[0.692516726,0.060687774,-0.040025666,0.717729422],[0,0,0,0],[9E+09,9E+09,9E+09,9E+09,9E+09,9E+09]];
    CONST robtarget Target_4460:=[[171.777441678,101.81849981,27.656565517],[0.692516726,0.060687774,-0.040025667,0.717729422],[0,0,0,0],[9E+09,9E+09,9E+09,9E+09,9E+09,9E+09]];
    CONST robtarget Target_4470:=[[171.544560342,101.396530417,27.661749925],[0.692516726,0.060687774,-0.040025666,0.717729422],[0,0,0,0],[9E+09,9E+09,9E+09,9E+09,9E+09,9E+09]];
    CONST robtarget Target_4480:=[[171.357610278,100.955786428,27.665660835],[0.692516726,0.060687774,-0.040025666,0.717729422],[0,0,0,0],[9E+09,9E+09,9E+09,9E+09,9E+09,9E+09]];
    CONST robtarget Target_4490:=[[171.216591489,100.496267845,27.668298248],[0.692516726,0.060687774,-0.040025666,0.717729422],[0,0,0,0],[9E+09,9E+09,9E+09,9E+09,9E+09,9E+09]];
    CONST robtarget Target_4500:=[[171.121503974,100.017974664,27.669662162],[0.692516726,0.060687774,-0.040025667,0.717729422],[0,0,0,0],[9E+09,9E+09,9E+09,9E+09,9E+09,9E+09]];
    CONST robtarget Target_4510:=[[171.072347734,99.520906889,27.669752579],[0.692516726,0.060687774,-0.040025666,0.717729422],[0,0,0,0],[9E+09,9E+09,9E+09,9E+09,9E+09,9E+09]];
    CONST robtarget Target_4520:=[[171.069122767,99.005064518,27.668569498],[0.692516726,0.060687774,-0.040025667,0.717729422],[0,0,0,0],[9E+09,9E+09,9E+09,9E+09,9E+09,9E+09]];
    CONST robtarget Target_4530:=[[171.492081286,87.751628834,27.629578293],[0.692516726,0.060687774,-0.040025667,0.717729422],[0,0,0,0],[9E+09,9E+09,9E+09,9E+09,9E+09,9E+09]];
    CONST robtarget Target_4540:=[[171.522569722,87.459846796,27.628045687],[0.692516726,0.060687774,-0.040025667,0.717729422],[0,0,0,0],[9E+09,9E+09,9E+09,9E+09,9E+09,9E+09]];
    CONST robtarget Target_4550:=[[171.590580768,87.208535937,27.625610043],[0.692516726,0.060687774,-0.040025666,0.717729422],[0,0,0,0],[9E+09,9E+09,9E+09,9E+09,9E+09,9E+09]];
    CONST robtarget Target_4560:=[[171.696114425,86.997696253,27.622271361],[0.692516726,0.060687774,-0.040025666,0.717729422],[0,0,0,0],[9E+09,9E+09,9E+09,9E+09,9E+09,9E+09]];
    CONST robtarget Target_4570:=[[171.839170691,86.827327746,27.61802964],[0.692516726,0.060687774,-0.040025667,0.717729422],[0,0,0,0],[9E+09,9E+09,9E+09,9E+09,9E+09,9E+09]];
    CONST robtarget Target_4580:=[[172.019749569,86.697430415,27.612884882],[0.692516726,0.060687774,-0.040025666,0.717729422],[0,0,0,0],[9E+09,9E+09,9E+09,9E+09,9E+09,9E+09]];
    CONST robtarget Target_4590:=[[172.237851057,86.608004262,27.606837086],[0.692516726,0.060687774,-0.040025666,0.717729422],[0,0,0,0],[9E+09,9E+09,9E+09,9E+09,9E+09,9E+09]];
    CONST robtarget Target_4600:=[[172.493475154,86.559049285,27.599886252],[0.692516726,0.060687774,-0.040025666,0.717729422],[0,0,0,0],[9E+09,9E+09,9E+09,9E+09,9E+09,9E+09]];
    CONST robtarget Target_4610:=[[172.786621862,86.550565484,27.59203238],[0.692516726,0.060687774,-0.040025667,0.717729422],[0,0,0,0],[9E+09,9E+09,9E+09,9E+09,9E+09,9E+09]];
    CONST robtarget Target_4620:=[[179.024782128,86.78560124,27.425924555],[0.692516726,0.060687774,-0.040025667,0.717729422],[0,0,0,0],[9E+09,9E+09,9E+09,9E+09,9E+09,9E+09]];
    CONST robtarget Target_4630:=[[179.538743807,86.827586588,27.4122946],[0.692516726,0.060687774,-0.040025667,0.717729422],[0,0,0,0],[9E+09,9E+09,9E+09,9E+09,9E+09,9E+09]];
    CONST robtarget Target_4640:=[[180.030538532,86.913978276,27.399366219],[0.692516726,0.060687774,-0.040025667,0.717729422],[0,0,0,0],[9E+09,9E+09,9E+09,9E+09,9E+09,9E+09]];
    CONST robtarget Target_4650:=[[180.500166302,87.044776303,27.387139411],[0.692516726,0.060687774,-0.040025667,0.717729422],[0,0,0,0],[9E+09,9E+09,9E+09,9E+09,9E+09,9E+09]];
    CONST robtarget Target_4660:=[[180.947627118,87.219980673,27.375614177],[0.692516726,0.060687774,-0.040025667,0.717729422],[0,0,0,0],[9E+09,9E+09,9E+09,9E+09,9E+09,9E+09]];
    CONST robtarget Target_4670:=[[181.37292098,87.439591383,27.364790517],[0.692516726,0.060687774,-0.040025667,0.717729422],[0,0,0,0],[9E+09,9E+09,9E+09,9E+09,9E+09,9E+09]];
    CONST robtarget Target_4680:=[[181.776047888,87.703608435,27.35466843],[0.692516726,0.060687774,-0.040025666,0.717729422],[0,0,0,0],[9E+09,9E+09,9E+09,9E+09,9E+09,9E+09]];
    CONST robtarget Target_4690:=[[182.157007841,88.012031827,27.345247917],[0.692516726,0.060687774,-0.040025666,0.717729422],[0,0,0,0],[9E+09,9E+09,9E+09,9E+09,9E+09,9E+09]];
    CONST robtarget Target_4700:=[[182.51580084,88.36486156,27.336528978],[0.692516726,0.060687774,-0.040025666,0.717729422],[0,0,0,0],[9E+09,9E+09,9E+09,9E+09,9E+09,9E+09]];
    CONST robtarget Target_4710:=[[182.840544726,88.749281761,27.328797574],[0.692516726,0.060687774,-0.040025666,0.717729422],[0,0,0,0],[9E+09,9E+09,9E+09,9E+09,9E+09,9E+09]];
    CONST robtarget Target_4720:=[[183.119357337,89.152476558,27.322339669],[0.692516726,0.060687774,-0.040025667,0.717729422],[0,0,0,0],[9E+09,9E+09,9E+09,9E+09,9E+09,9E+09]];
    CONST robtarget Target_4730:=[[183.352238674,89.574445951,27.317155261],[0.692516726,0.060687774,-0.040025666,0.717729422],[0,0,0,0],[9E+09,9E+09,9E+09,9E+09,9E+09,9E+09]];
    CONST robtarget Target_4740:=[[183.539188736,90.015189939,27.313244351],[0.692516726,0.060687774,-0.040025666,0.717729422],[0,0,0,0],[9E+09,9E+09,9E+09,9E+09,9E+09,9E+09]];
    CONST robtarget Target_4750:=[[183.680207525,90.474708523,27.310606938],[0.692516726,0.060687774,-0.040025666,0.717729422],[0,0,0,0],[9E+09,9E+09,9E+09,9E+09,9E+09,9E+09]];
    CONST robtarget Target_4760:=[[183.775295041,90.953001704,27.309243024],[0.692516726,0.060687774,-0.040025667,0.717729422],[0,0,0,0],[9E+09,9E+09,9E+09,9E+09,9E+09,9E+09]];
    CONST robtarget Target_4770:=[[183.824451281,91.450069479,27.309152607],[0.692516726,0.060687774,-0.040025666,0.717729422],[0,0,0,0],[9E+09,9E+09,9E+09,9E+09,9E+09,9E+09]];
    CONST robtarget Target_4780:=[[183.827676248,91.96591185,27.310335688],[0.692516726,0.060687774,-0.040025667,0.717729422],[0,0,0,0],[9E+09,9E+09,9E+09,9E+09,9E+09,9E+09]];
    CONST robtarget Target_4790:=[[183.805009768,92.300626295,27.311764925],[0.692516726,0.060687774,-0.040025667,0.717729422],[0,0,0,0],[9E+09,9E+09,9E+09,9E+09,9E+09,9E+09]];
    CONST robtarget Target_4800:=[[183.762419114,92.628731438,27.313710282],[0.692516726,0.060687774,-0.040025666,0.717729422],[0,0,0,0],[9E+09,9E+09,9E+09,9E+09,9E+09,9E+09]];
    CONST robtarget Target_4810:=[[183.699904283,92.950227282,27.316171758],[0.692516726,0.060687774,-0.040025666,0.717729422],[0,0,0,0],[9E+09,9E+09,9E+09,9E+09,9E+09,9E+09]];
    CONST robtarget Target_4820:=[[183.617465277,93.265113825,27.319149354],[0.692516726,0.060687774,-0.040025666,0.717729422],[0,0,0,0],[9E+09,9E+09,9E+09,9E+09,9E+09,9E+09]];
    CONST robtarget Target_4830:=[[183.515102095,93.573391069,27.322643069],[0.692516726,0.060687774,-0.040025667,0.717729422],[0,0,0,0],[9E+09,9E+09,9E+09,9E+09,9E+09,9E+09]];
    CONST robtarget Target_4840:=[[183.392814739,93.875059013,27.326652904],[0.692516726,0.060687774,-0.040025667,0.717729422],[0,0,0,0],[9E+09,9E+09,9E+09,9E+09,9E+09,9E+09]];
    CONST robtarget Target_4850:=[[183.250603206,94.170117656,27.331178858],[0.692516726,0.060687774,-0.040025667,0.717729422],[0,0,0,0],[9E+09,9E+09,9E+09,9E+09,9E+09,9E+09]];
    CONST robtarget Target_4860:=[[183.088467499,94.458566999,27.336220932],[0.692516726,0.060687774,-0.040025667,0.717729422],[0,0,0,0],[9E+09,9E+09,9E+09,9E+09,9E+09,9E+09]];
    CONST robtarget Target_4870:=[[182.892087356,94.751340618,27.34218867],[0.692516726,0.060687774,-0.040025666,0.717729422],[0,0,0,0],[9E+09,9E+09,9E+09,9E+09,9E+09,9E+09]];
    CONST robtarget Target_4880:=[[182.684899952,95.024341073,27.348396531],[0.692516726,0.060687774,-0.040025667,0.717729422],[0,0,0,0],[9E+09,9E+09,9E+09,9E+09,9E+09,9E+09]];
    CONST robtarget Target_4890:=[[182.466905288,95.277568363,27.354844512],[0.692516726,0.060687774,-0.040025667,0.717729422],[0,0,0,0],[9E+09,9E+09,9E+09,9E+09,9E+09,9E+09]];
    CONST robtarget Target_4900:=[[182.238103364,95.511022491,27.361532616],[0.692516726,0.060687774,-0.040025666,0.717729422],[0,0,0,0],[9E+09,9E+09,9E+09,9E+09,9E+09,9E+09]];
    CONST robtarget Target_4910:=[[181.998494178,95.724703455,27.368460841],[0.692516726,0.060687774,-0.040025667,0.717729422],[0,0,0,0],[9E+09,9E+09,9E+09,9E+09,9E+09,9E+09]];
    CONST robtarget Target_4920:=[[181.748077733,95.918611254,27.375629187],[0.692516726,0.060687774,-0.040025667,0.717729422],[0,0,0,0],[9E+09,9E+09,9E+09,9E+09,9E+09,9E+09]];
    CONST robtarget Target_4930:=[[181.486854027,96.09274589,27.383037656],[0.692516726,0.060687774,-0.040025667,0.717729422],[0,0,0,0],[9E+09,9E+09,9E+09,9E+09,9E+09,9E+09]];
    CONST robtarget Target_4940:=[[181.21482306,96.247107363,27.390686245],[0.692516726,0.060687774,-0.040025667,0.717729422],[0,0,0,0],[9E+09,9E+09,9E+09,9E+09,9E+09,9E+09]];
    CONST robtarget Target_4950:=[[180.931984832,96.381695672,27.398574957],[0.692516726,0.060687774,-0.040025667,0.717729422],[0,0,0,0],[9E+09,9E+09,9E+09,9E+09,9E+09,9E+09]];
    CONST robtarget Target_4960:=[[180.638339343,96.496510817,27.40670379],[0.692516726,0.060687774,-0.040025666,0.717729422],[0,0,0,0],[9E+09,9E+09,9E+09,9E+09,9E+09,9E+09]];
    CONST robtarget Target_4970:=[[180.333886595,96.591552798,27.415072744],[0.692516726,0.060687774,-0.040025666,0.717729422],[0,0,0,0],[9E+09,9E+09,9E+09,9E+09,9E+09,9E+09]];
    CONST robtarget Target_4980:=[[180.018626586,96.666821616,27.42368182],[0.692516726,0.060687774,-0.040025667,0.717729422],[0,0,0,0],[9E+09,9E+09,9E+09,9E+09,9E+09,9E+09]];
    CONST robtarget Target_4990:=[[179.692559316,96.722317269,27.432531018],[0.692516726,0.060687774,-0.040025666,0.717729422],[0,0,0,0],[9E+09,9E+09,9E+09,9E+09,9E+09,9E+09]];
    CONST robtarget Target_5000:=[[179.355684785,96.75803976,27.441620337],[0.692516726,0.060687774,-0.040025667,0.717729422],[0,0,0,0],[9E+09,9E+09,9E+09,9E+09,9E+09,9E+09]];
    CONST robtarget Target_5010:=[[179.008002993,96.773989085,27.450949778],[0.692516726,0.060687774,-0.040025667,0.717729422],[0,0,0,0],[9E+09,9E+09,9E+09,9E+09,9E+09,9E+09]];
    CONST robtarget Target_5020:=[[178.649513941,96.770165249,27.46051934],[0.692516726,0.060687774,-0.040025667,0.717729422],[0,0,0,0],[9E+09,9E+09,9E+09,9E+09,9E+09,9E+09]];
    CONST robtarget Target_5030:=[[173.658985729,96.582136643,27.5934056],[0.692516726,0.060687774,-0.040025667,0.717729422],[0,0,0,0],[9E+09,9E+09,9E+09,9E+09,9E+09,9E+09]];
    CONST robtarget Target_5040:=[[173.564386874,99.09907882,27.602126368],[0.692516726,0.060687774,-0.040025667,0.717729422],[0,0,0,0],[9E+09,9E+09,9E+09,9E+09,9E+09,9E+09]];
    CONST robtarget Target_5050:=[[172.763063297,99.172868608,-2.38707895],[0.692516726,0.060687774,-0.040025667,0.717729422],[0,0,0,0],[9E+09,9E+09,9E+09,9E+09,9E+09,9E+09]];
    CONST robtarget Target_5060:=[[232.681860655,69.262609655,-4.061728749],[0.692516726,0.060687774,-0.040025667,0.717729422],[-2,0,-1,0],[9E+09,9E+09,9E+09,9E+09,9E+09,9E+09]];
    CONST robtarget Target_5070:=[[233.483184232,69.188819867,25.927476569],[0.692516726,0.060687774,-0.040025667,0.717729422],[-2,0,-1,0],[9E+09,9E+09,9E+09,9E+09,9E+09,9E+09]];
    CONST robtarget Target_5080:=[[233.190037524,69.197303668,25.935330441],[0.692516726,0.060687774,-0.040025666,0.717729422],[-2,0,-1,0],[9E+09,9E+09,9E+09,9E+09,9E+09,9E+09]];
    CONST robtarget Target_5090:=[[232.934413426,69.246258645,25.942281275],[0.692516726,0.060687774,-0.040025666,0.717729422],[-2,0,-1,0],[9E+09,9E+09,9E+09,9E+09,9E+09,9E+09]];
    CONST robtarget Target_5100:=[[232.716311938,69.335684799,25.948329071],[0.692516726,0.060687774,-0.040025666,0.717729422],[-1,-1,0,0],[9E+09,9E+09,9E+09,9E+09,9E+09,9E+09]];
    CONST robtarget Target_5110:=[[232.535733061,69.465582129,25.953473829],[0.692516726,0.060687774,-0.040025667,0.717729422],[-1,-1,0,0],[9E+09,9E+09,9E+09,9E+09,9E+09,9E+09]];
    CONST robtarget Target_5120:=[[232.392676794,69.635950636,25.957715549],[0.692516726,0.060687774,-0.040025666,0.717729422],[-1,-1,0,0],[9E+09,9E+09,9E+09,9E+09,9E+09,9E+09]];
    CONST robtarget Target_5130:=[[232.287143138,69.84679032,25.961054231],[0.692516726,0.060687774,-0.040025666,0.717729422],[-1,-1,0,0],[9E+09,9E+09,9E+09,9E+09,9E+09,9E+09]];
    CONST robtarget Target_5140:=[[232.219132091,70.09810118,25.963489876],[0.692516726,0.060687774,-0.040025667,0.717729422],[-1,-1,0,0],[9E+09,9E+09,9E+09,9E+09,9E+09,9E+09]];
    CONST robtarget Target_5150:=[[232.188643656,70.389883217,25.965022482],[0.692516726,0.060687774,-0.040025667,0.717729422],[-1,-1,0,0],[9E+09,9E+09,9E+09,9E+09,9E+09,9E+09]];
    CONST robtarget Target_5160:=[[232.197143721,70.683134228,25.965516914],[0.692516726,0.060687774,-0.040025667,0.717729422],[-1,-1,0,0],[9E+09,9E+09,9E+09,9E+09,9E+09,9E+09]];
    CONST robtarget Target_5170:=[[232.24609818,70.938852008,25.964838036],[0.692516726,0.060687774,-0.040025666,0.717729422],[-1,-1,0,0],[9E+09,9E+09,9E+09,9E+09,9E+09,9E+09]];
    CONST robtarget Target_5180:=[[232.335507031,71.157036559,25.962985849],[0.692516726,0.060687774,-0.040025667,0.717729422],[-1,-1,0,0],[9E+09,9E+09,9E+09,9E+09,9E+09,9E+09]];
    CONST robtarget Target_5190:=[[232.465370276,71.337687881,25.959960351],[0.692516726,0.060687774,-0.040025666,0.717729422],[-1,-1,0,0],[9E+09,9E+09,9E+09,9E+09,9E+09,9E+09]];
    CONST robtarget Target_5200:=[[232.635687914,71.480805972,25.955761544],[0.692516726,0.060687774,-0.040025667,0.717729422],[-1,-1,0,0],[9E+09,9E+09,9E+09,9E+09,9E+09,9E+09]];
    CONST robtarget Target_5210:=[[232.846459945,71.586390835,25.950389428],[0.692516726,0.060687774,-0.040025667,0.717729422],[-1,-1,0,0],[9E+09,9E+09,9E+09,9E+09,9E+09,9E+09]];
    CONST robtarget Target_5220:=[[233.097686369,71.654442466,25.943844001],[0.692516726,0.060687774,-0.040025666,0.717729422],[-1,-1,0,0],[9E+09,9E+09,9E+09,9E+09,9E+09,9E+09]];
    CONST robtarget Target_5230:=[[233.389367185,71.68496087,25.936125265],[0.692516726,0.060687774,-0.040025667,0.717729422],[-2,0,-1,0],[9E+09,9E+09,9E+09,9E+09,9E+09,9E+09]];
    CONST robtarget Target_5240:=[[240.895953372,71.96778723,25.736242182],[0.692516726,0.060687774,-0.040025667,0.717729422],[-2,0,-1,0],[9E+09,9E+09,9E+09,9E+09,9E+09,9E+09]];
    CONST robtarget Target_5250:=[[241.529941703,71.96303195,25.71929006],[0.692516726,0.060687774,-0.040025667,0.717729422],[-2,0,-1,0],[9E+09,9E+09,9E+09,9E+09,9E+09,9E+09]];
    CONST robtarget Target_5260:=[[242.142686907,71.900192055,25.702762642],[0.692516726,0.060687774,-0.040025666,0.717729422],[-2,0,-1,0],[9E+09,9E+09,9E+09,9E+09,9E+09,9E+09]];
    CONST robtarget Target_5270:=[[242.734188983,71.779267546,25.68665993],[0.692516726,0.060687774,-0.040025667,0.717729422],[-2,0,-1,0],[9E+09,9E+09,9E+09,9E+09,9E+09,9E+09]];
    CONST robtarget Target_5280:=[[243.304447933,71.60025842,25.670981922],[0.692516726,0.060687774,-0.040025666,0.717729422],[-2,0,-1,0],[9E+09,9E+09,9E+09,9E+09,9E+09,9E+09]];
    CONST robtarget Target_5290:=[[243.853463755,71.363164679,25.65572862],[0.692516726,0.060687774,-0.040025667,0.717729422],[-2,0,-1,0],[9E+09,9E+09,9E+09,9E+09,9E+09,9E+09]];
    CONST robtarget Target_5300:=[[244.381236451,71.067986322,25.640900022],[0.692516726,0.060687774,-0.040025667,0.717729422],[-2,0,-1,0],[9E+09,9E+09,9E+09,9E+09,9E+09,9E+09]];
    CONST robtarget Target_5310:=[[244.88776602,70.71472335,25.62649613],[0.692516726,0.060687774,-0.040025667,0.717729422],[-2,0,-1,0],[9E+09,9E+09,9E+09,9E+09,9E+09,9E+09]];
    CONST robtarget Target_5320:=[[245.373052462,70.303375763,25.612516942],[0.692516726,0.060687774,-0.040025667,0.717729422],[-2,0,-1,0],[9E+09,9E+09,9E+09,9E+09,9E+09,9E+09]];
    CONST robtarget Target_5330:=[[245.819565539,69.85020796,25.599470894],[0.692516726,0.060687774,-0.040025666,0.717729422],[-2,0,-1,0],[9E+09,9E+09,9E+09,9E+09,9E+09,9E+09]];
    CONST robtarget Target_5340:=[[246.209775016,69.371484341,25.58786642],[0.692516726,0.060687774,-0.040025667,0.717729422],[-2,0,-1,0],[9E+09,9E+09,9E+09,9E+09,9E+09,9E+09]];
    CONST robtarget Target_5350:=[[246.543680891,68.867204905,25.577703519],[0.692516726,0.060687774,-0.040025666,0.717729422],[-2,0,-1,0],[9E+09,9E+09,9E+09,9E+09,9E+09,9E+09]];
    CONST robtarget Target_5360:=[[246.821283166,68.337369653,25.568982192],[0.692516726,0.060687774,-0.040025666,0.717729422],[-2,0,-1,0],[9E+09,9E+09,9E+09,9E+09,9E+09,9E+09]];
    CONST robtarget Target_5370:=[[247.04258184,67.781978585,25.561702438],[0.692516726,0.060687774,-0.040025666,0.717729422],[-2,0,-1,0],[9E+09,9E+09,9E+09,9E+09,9E+09,9E+09]];
    CONST robtarget Target_5380:=[[247.207576913,67.2010317,25.555864257],[0.692516726,0.060687774,-0.040025666,0.717729422],[-2,0,-1,0],[9E+09,9E+09,9E+09,9E+09,9E+09,9E+09]];
    CONST robtarget Target_5390:=[[247.316268385,66.594528999,25.551467651],[0.692516726,0.060687774,-0.040025667,0.717729422],[-2,0,-1,0],[9E+09,9E+09,9E+09,9E+09,9E+09,9E+09]];
    CONST robtarget Target_5400:=[[247.368656255,65.962470481,25.548512617],[0.692516726,0.060687774,-0.040025667,0.717729422],[-2,0,-1,0],[9E+09,9E+09,9E+09,9E+09,9E+09,9E+09]];
    CONST robtarget Target_5410:=[[247.838523297,53.460964297,25.505197064],[0.692516726,0.060687774,-0.040025667,0.717729422],[-2,0,-1,0],[9E+09,9E+09,9E+09,9E+09,9E+09,9E+09]];
    CONST robtarget Target_5420:=[[247.833728033,52.826751286,25.503764686],[0.692516726,0.060687774,-0.040025666,0.717729422],[-2,0,-1,0],[9E+09,9E+09,9E+09,9E+09,9E+09,9E+09]];
    CONST robtarget Target_5430:=[[247.770870098,52.213785101,25.503936044],[0.692516726,0.060687774,-0.040025667,0.717729422],[-2,0,-1,0],[9E+09,9E+09,9E+09,9E+09,9E+09,9E+09]];
    CONST robtarget Target_5440:=[[247.649949491,51.622065745,25.505711139],[0.692516726,0.060687774,-0.040025667,0.717729422],[-2,0,-1,0],[9E+09,9E+09,9E+09,9E+09,9E+09,9E+09]];
    CONST robtarget Target_5450:=[[247.470966214,51.051593215,25.50908997],[0.692516726,0.060687774,-0.040025667,0.717729422],[-2,0,-1,0],[9E+09,9E+09,9E+09,9E+09,9E+09,9E+09]];
    CONST robtarget Target_5460:=[[247.233920267,50.502367513,25.514072538],[0.692516726,0.060687774,-0.040025666,0.717729422],[-2,0,-1,0],[9E+09,9E+09,9E+09,9E+09,9E+09,9E+09]];
    CONST robtarget Target_5470:=[[246.93881165,49.974388638,25.520658843],[0.692516726,0.060687774,-0.040025667,0.717729422],[-2,0,-1,0],[9E+09,9E+09,9E+09,9E+09,9E+09,9E+09]];
    CONST robtarget Target_5480:=[[246.585640361,49.467656591,25.528848884],[0.692516726,0.060687774,-0.040025667,0.717729422],[-2,0,-1,0],[9E+09,9E+09,9E+09,9E+09,9E+09,9E+09]];
    CONST robtarget Target_5490:=[[246.174406402,48.982171371,25.538642662],[0.692516726,0.060687774,-0.040025666,0.717729422],[-2,0,-1,0],[9E+09,9E+09,9E+09,9E+09,9E+09,9E+09]];
    CONST robtarget Target_5500:=[[245.72136957,48.535470489,25.54964886],[0.692516726,0.060687774,-0.040025666,0.717729422],[-2,0,-1,0],[9E+09,9E+09,9E+09,9E+09,9E+09,9E+09]];
    CONST robtarget Target_5510:=[[245.242789664,48.145091454,25.561476162],[0.692516726,0.060687774,-0.040025667,0.717729422],[-2,0,-1,0],[9E+09,9E+09,9E+09,9E+09,9E+09,9E+09]];
    CONST robtarget Target_5520:=[[244.738666681,47.811034267,25.574124567],[0.692516726,0.060687774,-0.040025666,0.717729422],[-2,0,-1,0],[9E+09,9E+09,9E+09,9E+09,9E+09,9E+09]];
    CONST robtarget Target_5530:=[[244.209000625,47.533298926,25.587594076],[0.692516726,0.060687774,-0.040025666,0.717729422],[-2,0,-1,0],[9E+09,9E+09,9E+09,9E+09,9E+09,9E+09]];
    CONST robtarget Target_5540:=[[243.653791493,47.311885433,25.601884689],[0.692516726,0.060687774,-0.040025666,0.717729422],[-2,0,-1,0],[9E+09,9E+09,9E+09,9E+09,9E+09,9E+09]];
    CONST robtarget Target_5550:=[[243.073039287,47.146793787,25.616996405],[0.692516726,0.060687774,-0.040025666,0.717729422],[-2,0,-1,0],[9E+09,9E+09,9E+09,9E+09,9E+09,9E+09]];
    CONST robtarget Target_5560:=[[242.466744005,47.038023987,25.632929225],[0.692516726,0.060687774,-0.040025667,0.717729422],[-2,0,-1,0],[9E+09,9E+09,9E+09,9E+09,9E+09,9E+09]];
